//     Term 99 (AT2000-0250)/CC Inputs/Current actual value Ch.3 <-> Data Pointer/CurrentActualValues[2]
//     Term 99 (AT2000-0250)/CC Inputs/Current actual value Ch.4 <-> Data Pointer/CurrentActualValues[3]
//     Term 99 (AT2000-0250)/CC Inputs/Current actual value Ch.5 <-> Data Pointer/CurrentActualValues[4]
//     Term 99 (AT2000-0250)/CC Inputs/Current actual value Ch.6 <-> Data Pointer/CurrentActualValues[5]
//     Term 99 (AT2000-0250)/CC Inputs/Current actual value Ch.7 <-> Data Pointer/CurrentActualValues[6]
//     Term 99 (AT2000-0250)/CC Inputs/Current actual value Ch.8 <-> Data Pointer/CurrentActualValues[7]
//     Term 99 (AT2000-0250)/CC Inputs/Current actual value Ch.9 <-> Data Pointer/CurrentActualValues[8]
//     Term 99 (AT2000-0250)/CC Inputs/Status <-> Data Pointer/Status
//     Term 99 (AT2000-0250)/CC Outputs/Control <-> Data Pointer/Control
//     Term 99 (AT2000-0250)/CC Outputs/Current setpoint value Ch.1 <-> Data Pointer/CurrentSetpointValues[0]
//     Term 99 (AT2000-0250)/CC Outputs/Current setpoint value Ch.10 <-> Data Pointer/CurrentSetpointValues[9]
//     Term 99 (AT2000-0250)/CC Outputs/Current setpoint value Ch.11 <-> Data Pointer/CurrentSetpointValues[10]
//     Term 99 (AT2000-0250)/CC Outputs/Current setpoint value Ch.12 <-> Data Pointer/CurrentSetpointValues[11]
//     Term 99 (AT2000-0250)/CC Outputs/Current setpoint value Ch.13 <-> Data Pointer/CurrentSetpointValues[12]
//     Term 99 (AT2000-0250)/CC Outputs/Current setpoint value Ch.14 <-> Data Pointer/CurrentSetpointValues[13]
//     Term 99 (AT2000-0250)/CC Outputs/Current setpoint value Ch.15 <-> Data Pointer/CurrentSetpointValues[14]
//     Term 99 (AT2000-0250)/CC Outputs/Current setpoint value Ch.2 <-> Data Pointer/CurrentSetpointValues[1]
//     Term 99 (AT2000-0250)/CC Outputs/Current setpoint value Ch.3 <-> Data Pointer/CurrentSetpointValues[2]
//     Term 99 (AT2000-0250)/CC Outputs/Current setpoint value Ch.4 <-> Data Pointer/CurrentSetpointValues[3]
//     Term 99 (AT2000-0250)/CC Outputs/Current setpoint value Ch.5 <-> Data Pointer/CurrentSetpointValues[4]
//     Term 99 (AT2000-0250)/CC Outputs/Current setpoint value Ch.6 <-> Data Pointer/CurrentSetpointValues[5]
//     Term 99 (AT2000-0250)/CC Outputs/Current setpoint value Ch.7 <-> Data Pointer/CurrentSetpointValues[6]
//     Term 99 (AT2000-0250)/CC Outputs/Current setpoint value Ch.8 <-> Data Pointer/CurrentSetpointValues[7]
//     Term 99 (AT2000-0250)/CC Outputs/Current setpoint value Ch.9 <-> Data Pointer/CurrentSetpointValues[8]
//     Term 99 (AT2000-0250)/Term 100 (AT2000-5250)/FB Inputs/Value Channel 01 <-> Data Pointer/RawPositionValues[0]
//     Term 99 (AT2000-0250)/Term 100 (AT2000-5250)/FB Inputs/Value Channel 02 <-> Data Pointer/RawPositionValues[1]
//     Term 99 (AT2000-0250)/Term 100 (AT2000-5250)/FB Inputs/Value Channel 03 <-> Data Pointer/RawPositionValues[2]
//     Term 99 (AT2000-0250)/Term 100 (AT2000-5250)/FB Inputs/Value Channel 04 <-> Data Pointer/RawPositionValues[3]
//     Term 99 (AT2000-0250)/Term 100 (AT2000-5250)/FB Inputs/Value Channel 05 <-> Data Pointer/RawPositionValues[4]
//     Term 99 (AT2000-0250)/Term 100 (AT2000-5250)/FB Inputs/Value Channel 06 <-> Data Pointer/RawPositionValues[5]
//     Term 99 (AT2000-0250)/Term 100 (AT2000-5250)/FB Inputs/Value Channel 07 <-> Data Pointer/RawPositionValues[6]
//     Term 99 (AT2000-0250)/Term 100 (AT2000-5250)/FB Inputs/Value Channel 08 <-> Data Pointer/RawPositionValues[7]
//     Term 99 (AT2000-0250)/Term 100 (AT2000-5250)/FB Inputs/Value Channel 09 <-> Data Pointer/RawPositionValues[8]
//     Term 99 (AT2000-0250)/Term 100 (AT2000-5250)/FB Inputs/Value Channel 10 <-> Data Pointer/RawPositionValues[9]
//     Term 99 (AT2000-0250)/Term 100 (AT2000-5250)/FB Inputs/Value Channel 11 <-> Data Pointer/RawPositionValues[10]
//     Term 99 (AT2000-0250)/Term 100 (AT2000-5250)/FB Inputs/Value Channel 12 <-> Data Pointer/RawPositionValues[11]
//     Term 99 (AT2000-0250)/Term 100 (AT2000-5250)/FB Inputs/Value Channel 13 <-> Data Pointer/RawPositionValues[12]
//     Term 99 (AT2000-0250)/Term 100 (AT2000-5250)/FB Inputs/Value Channel 14 <-> Data Pointer/RawPositionValues[13]
//     Term 99 (AT2000-0250)/Term 100 (AT2000-5250)/FB Inputs/Value Channel 15 <-> Data Pointer/RawPositionValues[14]
//     Term 99 (AT2000-0250)/Term 100 (AT2000-5250)/FB Inputs/Value Channel 16 <-> Data Pointer/RawPositionValues[15]
//     Term 99 (AT2000-0250)/Term 100 (AT2000-5250)/FB Inputs/Value Channel 17 <-> Data Pointer/RawPositionValues[16]
//     Term 99 (AT2000-0250)/Term 100 (AT2000-5250)/FB Inputs/Value Channel 18 <-> Data Pointer/RawPositionValues[17]
//     Term 99 (AT2000-0250)/Term 100 (AT2000-5250)/FB Inputs/Value Channel 19 <-> Data Pointer/RawPositionValues[18]
//     Term 99 (AT2000-0250)/Term 100 (AT2000-5250)/FB Inputs/Value Channel 20 <-> Data Pointer/RawPositionValues[19]
//     Term 99 (AT2000-0250)/Term 100 (AT2000-5250)/FB Inputs/Value Channel 21 <-> Data Pointer/RawPositionValues[20]
//     Term 99 (AT2000-0250)/Term 100 (AT2000-5250)/FB Inputs/Value Channel 22 <-> Data Pointer/RawPositionValues[21]
//     Term 99 (AT2000-0250)/Term 100 (AT2000-5250)/FB Inputs/Value Channel 23 <-> Data Pointer/RawPositionValues[22]
//     Term 99 (AT2000-0250)/Term 100 (AT2000-5250)/FB Inputs/Value Channel 24 <-> Data Pointer/RawPositionValues[23]
//     Term 99 (AT2000-0250)/Term 100 (AT2000-5250)/FB Inputs/Value Channel 25 <-> Data Pointer/RawPositionValues[24]
//     Term 99 (AT2000-0250)/Term 100 (AT2000-5250)/FB Inputs/Value Channel 26 <-> Data Pointer/RawPositionValues[25]
//     Term 99 (AT2000-0250)/Term 100 (AT2000-5250)/FB Inputs/Value Channel 27 <-> Data Pointer/RawPositionValues[26]
//     Term 99 (AT2000-0250)/Term 100 (AT2000-5250)/FB Inputs/Value Channel 28 <-> Data Pointer/RawPositionValues[27]
//     Term 99 (AT2000-0250)/Term 100 (AT2000-5250)/FB Inputs/Value Channel 29 <-> Data Pointer/RawPositionValues[28]
//     Term 99 (AT2000-0250)/Term 100 (AT2000-5250)/FB Inputs/Value Channel 30 <-> Data Pointer/RawPositionValues[29]
//     Term 99 (AT2000-0250)/Term 100 (AT2000-5250)/FB Inputs/Value Channel 31 <-> Data Pointer/RawPositionValues[30]
//     Term 99 (AT2000-0250)/Term 100 (AT2000-5250)/FB Inputs/Value Channel 32 <-> Data Pointer/RawPositionValues[31]
//   Device 23 <-> TcCOM Objects/XTS ProcessingUnit 1/Part 1/Module 51
//     Term 101 (AT2000-0250)/CC Inputs/Current actual value Ch.1 <-> Data Pointer/CurrentActualValues[0]
//     Term 101 (AT2000-0250)/CC Inputs/Current actual value Ch.10 <-> Data Pointer/CurrentActualValues[9]
//     Term 101 (AT2000-0250)/CC Inputs/Current actual value Ch.11 <-> Data Pointer/CurrentActualValues[10]
//     Term 101 (AT2000-0250)/CC Inputs/Current actual value Ch.12 <-> Data Pointer/CurrentActualValues[11]
//     Term 101 (AT2000-0250)/CC Inputs/Current actual value Ch.13 <-> Data Pointer/CurrentActualValues[12]
//     Term 101 (AT2000-0250)/CC Inputs/Current actual value Ch.14 <-> Data Pointer/CurrentActualValues[13]
//     Term 101 (AT2000-0250)/CC Inputs/Current actual value Ch.15 <-> Data Pointer/CurrentActualValues[14]
//     Term 101 (AT2000-0250)/CC Inputs/Current actual value Ch.2 <-> Data Pointer/CurrentActualValues[1]
//     Term 101 (AT2000-0250)/CC Inputs/Current actual value Ch.3 <-> Data Pointer/CurrentActualValues[2]
//     Term 101 (AT2000-0250)/CC Inputs/Current actual value Ch.4 <-> Data Pointer/CurrentActualValues[3]
//     Term 101 (AT2000-0250)/CC Inputs/Current actual value Ch.5 <-> Data Pointer/CurrentActualValues[4]
//     Term 101 (AT2000-0250)/CC Inputs/Current actual value Ch.6 <-> Data Pointer/CurrentActualValues[5]
//     Term 101 (AT2000-0250)/CC Inputs/Current actual value Ch.7 <-> Data Pointer/CurrentActualValues[6]
//     Term 101 (AT2000-0250)/CC Inputs/Current actual value Ch.8 <-> Data Pointer/CurrentActualValues[7]
//     Term 101 (AT2000-0250)/CC Inputs/Current actual value Ch.9 <-> Data Pointer/CurrentActualValues[8]
//     Term 101 (AT2000-0250)/CC Inputs/Status <-> Data Pointer/Status
//     Term 101 (AT2000-0250)/CC Outputs/Control <-> Data Pointer/Control
//     Term 101 (AT2000-0250)/CC Outputs/Current setpoint value Ch.1 <-> Data Pointer/CurrentSetpointValues[0]
//     Term 101 (AT2000-0250)/CC Outputs/Current setpoint value Ch.10 <-> Data Pointer/CurrentSetpointValues[9]
//     Term 101 (AT2000-0250)/CC Outputs/Current setpoint value Ch.11 <-> Data Pointer/CurrentSetpointValues[10]
//     Term 101 (AT2000-0250)/CC Outputs/Current setpoint value Ch.12 <-> Data Pointer/CurrentSetpointValues[11]
//     Term 101 (AT2000-0250)/CC Outputs/Current setpoint value Ch.13 <-> Data Pointer/CurrentSetpointValues[12]
//     Term 101 (AT2000-0250)/CC Outputs/Current setpoint value Ch.14 <-> Data Pointer/CurrentSetpointValues[13]
//     Term 101 (AT2000-0250)/CC Outputs/Current setpoint value Ch.15 <-> Data Pointer/CurrentSetpointValues[14]
//     Term 101 (AT2000-0250)/CC Outputs/Current setpoint value Ch.2 <-> Data Pointer/CurrentSetpointValues[1]
//     Term 101 (AT2000-0250)/CC Outputs/Current setpoint value Ch.3 <-> Data Pointer/CurrentSetpointValues[2]
//     Term 101 (AT2000-0250)/CC Outputs/Current setpoint value Ch.4 <-> Data Pointer/CurrentSetpointValues[3]
//     Term 101 (AT2000-0250)/CC Outputs/Current setpoint value Ch.5 <-> Data Pointer/CurrentSetpointValues[4]
//     Term 101 (AT2000-0250)/CC Outputs/Current setpoint value Ch.6 <-> Data Pointer/CurrentSetpointValues[5]
//     Term 101 (AT2000-0250)/CC Outputs/Current setpoint value Ch.7 <-> Data Pointer/CurrentSetpointValues[6]
//     Term 101 (AT2000-0250)/CC Outputs/Current setpoint value Ch.8 <-> Data Pointer/CurrentSetpointValues[7]
//     Term 101 (AT2000-0250)/CC Outputs/Current setpoint value Ch.9 <-> Data Pointer/CurrentSetpointValues[8]
//     Term 101 (AT2000-0250)/Term 102 (AT2000-5250)/FB Inputs/Value Channel 01 <-> Data Pointer/RawPositionValues[0]
//     Term 101 (AT2000-0250)/Term 102 (AT2000-5250)/FB Inputs/Value Channel 02 <-> Data Pointer/RawPositionValues[1]
//     Term 101 (AT2000-0250)/Term 102 (AT2000-5250)/FB Inputs/Value Channel 03 <-> Data Pointer/RawPositionValues[2]
//     Term 101 (AT2000-0250)/Term 102 (AT2000-5250)/FB Inputs/Value Channel 04 <-> Data Pointer/RawPositionValues[3]
//     Term 101 (AT2000-0250)/Term 102 (AT2000-5250)/FB Inputs/Value Channel 05 <-> Data Pointer/RawPositionValues[4]
//     Term 101 (AT2000-0250)/Term 102 (AT2000-5250)/FB Inputs/Value Channel 06 <-> Data Pointer/RawPositionValues[5]
//     Term 101 (AT2000-0250)/Term 102 (AT2000-5250)/FB Inputs/Value Channel 07 <-> Data Pointer/RawPositionValues[6]
//     Term 101 (AT2000-0250)/Term 102 (AT2000-5250)/FB Inputs/Value Channel 08 <-> Data Pointer/RawPositionValues[7]
//     Term 101 (AT2000-0250)/Term 102 (AT2000-5250)/FB Inputs/Value Channel 09 <-> Data Pointer/RawPositionValues[8]
//     Term 101 (AT2000-0250)/Term 102 (AT2000-5250)/FB Inputs/Value Channel 10 <-> Data Pointer/RawPositionValues[9]
//     Term 101 (AT2000-0250)/Term 102 (AT2000-5250)/FB Inputs/Value Channel 11 <-> Data Pointer/RawPositionValues[10]
//     Term 101 (AT2000-0250)/Term 102 (AT2000-5250)/FB Inputs/Value Channel 12 <-> Data Pointer/RawPositionValues[11]
//     Term 101 (AT2000-0250)/Term 102 (AT2000-5250)/FB Inputs/Value Channel 13 <-> Data Pointer/RawPositionValues[12]
//     Term 101 (AT2000-0250)/Term 102 (AT2000-5250)/FB Inputs/Value Channel 14 <-> Data Pointer/RawPositionValues[13]
//     Term 101 (AT2000-0250)/Term 102 (AT2000-5250)/FB Inputs/Value Channel 15 <-> Data Pointer/RawPositionValues[14]
//     Term 101 (AT2000-0250)/Term 102 (AT2000-5250)/FB Inputs/Value Channel 16 <-> Data Pointer/RawPositionValues[15]
//     Term 101 (AT2000-0250)/Term 102 (AT2000-5250)/FB Inputs/Value Channel 17 <-> Data Pointer/RawPositionValues[16]
//     Term 101 (AT2000-0250)/Term 102 (AT2000-5250)/FB Inputs/Value Channel 18 <-> Data Pointer/RawPositionValues[17]
//     Term 101 (AT2000-0250)/Term 102 (AT2000-5250)/FB Inputs/Value Channel 19 <-> Data Pointer/RawPositionValues[18]
//     Term 101 (AT2000-0250)/Term 102 (AT2000-5250)/FB Inputs/Value Channel 20 <-> Data Pointer/RawPositionValues[19]
//     Term 101 (AT2000-0250)/Term 102 (AT2000-5250)/FB Inputs/Value Channel 21 <-> Data Pointer/RawPositionValues[20]
//     Term 101 (AT2000-0250)/Term 102 (AT2000-5250)/FB Inputs/Value Channel 22 <-> Data Pointer/RawPositionValues[21]
//     Term 101 (AT2000-0250)/Term 102 (AT2000-5250)/FB Inputs/Value Channel 23 <-> Data Pointer/RawPositionValues[22]
//     Term 101 (AT2000-0250)/Term 102 (AT2000-5250)/FB Inputs/Value Channel 24 <-> Data Pointer/RawPositionValues[23]
//     Term 101 (AT2000-0250)/Term 102 (AT2000-5250)/FB Inputs/Value Channel 25 <-> Data Pointer/RawPositionValues[24]
//     Term 101 (AT2000-0250)/Term 102 (AT2000-5250)/FB Inputs/Value Channel 26 <-> Data Pointer/RawPositionValues[25]
//     Term 101 (AT2000-0250)/Term 102 (AT2000-5250)/FB Inputs/Value Channel 27 <-> Data Pointer/RawPositionValues[26]
//     Term 101 (AT2000-0250)/Term 102 (AT2000-5250)/FB Inputs/Value Channel 28 <-> Data Pointer/RawPositionValues[27]
//     Term 101 (AT2000-0250)/Term 102 (AT2000-5250)/FB Inputs/Value Channel 29 <-> Data Pointer/RawPositionValues[28]
//     Term 101 (AT2000-0250)/Term 102 (AT2000-5250)/FB Inputs/Value Channel 30 <-> Data Pointer/RawPositionValues[29]
//     Term 101 (AT2000-0250)/Term 102 (AT2000-5250)/FB Inputs/Value Channel 31 <-> Data Pointer/RawPositionValues[30]
//     Term 101 (AT2000-0250)/Term 102 (AT2000-5250)/FB Inputs/Value Channel 32 <-> Data Pointer/RawPositionValues[31]
//   Device 23 <-> TcCOM Objects/XTS ProcessingUnit 1/Part 1/Module 52
//     Term 103 (AT2000-0250)/CC Inputs/Current actual value Ch.1 <-> Data Pointer/CurrentActualValues[0]
//     Term 103 (AT2000-0250)/CC Inputs/Current actual value Ch.10 <-> Data Pointer/CurrentActualValues[9]
//     Term 103 (AT2000-0250)/CC Inputs/Current actual value Ch.11 <-> Data Pointer/CurrentActualValues[10]
//     Term 103 (AT2000-0250)/CC Inputs/Current actual value Ch.12 <-> Data Pointer/CurrentActualValues[11]
//     Term 103 (AT2000-0250)/CC Inputs/Current actual value Ch.13 <-> Data Pointer/CurrentActualValues[12]
//     Term 103 (AT2000-0250)/CC Inputs/Current actual value Ch.14 <-> Data Pointer/CurrentActualValues[13]
//     Term 103 (AT2000-0250)/CC Inputs/Current actual value Ch.15 <-> Data Pointer/CurrentActualValues[14]
//     Term 103 (AT2000-0250)/CC Inputs/Current actual value Ch.2 <-> Data Pointer/CurrentActualValues[1]
//     Term 103 (AT2000-0250)/CC Inputs/Current actual value Ch.3 <-> Data Pointer/CurrentActualValues[2]
//     Term 103 (AT2000-0250)/CC Inputs/Current actual value Ch.4 <-> Data Pointer/CurrentActualValues[3]
//     Term 103 (AT2000-0250)/CC Inputs/Current actual value Ch.5 <-> Data Pointer/CurrentActualValues[4]
//     Term 103 (AT2000-0250)/CC Inputs/Current actual value Ch.6 <-> Data Pointer/CurrentActualValues[5]
//     Term 103 (AT2000-0250)/CC Inputs/Current actual value Ch.7 <-> Data Pointer/CurrentActualValues[6]
//     Term 103 (AT2000-0250)/CC Inputs/Current actual value Ch.8 <-> Data Pointer/CurrentActualValues[7]
//     Term 103 (AT2000-0250)/CC Inputs/Current actual value Ch.9 <-> Data Pointer/CurrentActualValues[8]
//     Term 103 (AT2000-0250)/CC Inputs/Status <-> Data Pointer/Status
//     Term 103 (AT2000-0250)/CC Outputs/Control <-> Data Pointer/Control
//     Term 103 (AT2000-0250)/CC Outputs/Current setpoint value Ch.1 <-> Data Pointer/CurrentSetpointValues[0]
//     Term 103 (AT2000-0250)/CC Outputs/Current setpoint value Ch.10 <-> Data Pointer/CurrentSetpointValues[9]
//     Term 103 (AT2000-0250)/CC Outputs/Current setpoint value Ch.11 <-> Data Pointer/CurrentSetpointValues[10]
//     Term 103 (AT2000-0250)/CC Outputs/Current setpoint value Ch.12 <-> Data Pointer/CurrentSetpointValues[11]
//     Term 103 (AT2000-0250)/CC Outputs/Current setpoint value Ch.13 <-> Data Pointer/CurrentSetpointValues[12]
//     Term 103 (AT2000-0250)/CC Outputs/Current setpoint value Ch.14 <-> Data Pointer/CurrentSetpointValues[13]
//     Term 103 (AT2000-0250)/CC Outputs/Current setpoint value Ch.15 <-> Data Pointer/CurrentSetpointValues[14]
//     Term 103 (AT2000-0250)/CC Outputs/Current setpoint value Ch.2 <-> Data Pointer/CurrentSetpointValues[1]
//     Term 103 (AT2000-0250)/CC Outputs/Current setpoint value Ch.3 <-> Data Pointer/CurrentSetpointValues[2]
//     Term 103 (AT2000-0250)/CC Outputs/Current setpoint value Ch.4 <-> Data Pointer/CurrentSetpointValues[3]
//     Term 103 (AT2000-0250)/CC Outputs/Current setpoint value Ch.5 <-> Data Pointer/CurrentSetpointValues[4]
//     Term 103 (AT2000-0250)/CC Outputs/Current setpoint value Ch.6 <-> Data Pointer/CurrentSetpointValues[5]
//     Term 103 (AT2000-0250)/CC Outputs/Current setpoint value Ch.7 <-> Data Pointer/CurrentSetpointValues[6]
//     Term 103 (AT2000-0250)/CC Outputs/Current setpoint value Ch.8 <-> Data Pointer/CurrentSetpointValues[7]
//     Term 103 (AT2000-0250)/CC Outputs/Current setpoint value Ch.9 <-> Data Pointer/CurrentSetpointValues[8]
//     Term 103 (AT2000-0250)/Term 104 (AT2000-5250)/FB Inputs/Value Channel 01 <-> Data Pointer/RawPositionValues[0]
//     Term 103 (AT2000-0250)/Term 104 (AT2000-5250)/FB Inputs/Value Channel 02 <-> Data Pointer/RawPositionValues[1]
//     Term 103 (AT2000-0250)/Term 104 (AT2000-5250)/FB Inputs/Value Channel 03 <-> Data Pointer/RawPositionValues[2]
//     Term 103 (AT2000-0250)/Term 104 (AT2000-5250)/FB Inputs/Value Channel 04 <-> Data Pointer/RawPositionValues[3]
//     Term 103 (AT2000-0250)/Term 104 (AT2000-5250)/FB Inputs/Value Channel 05 <-> Data Pointer/RawPositionValues[4]
//     Term 103 (AT2000-0250)/Term 104 (AT2000-5250)/FB Inputs/Value Channel 06 <-> Data Pointer/RawPositionValues[5]
//     Term 103 (AT2000-0250)/Term 104 (AT2000-5250)/FB Inputs/Value Channel 07 <-> Data Pointer/RawPositionValues[6]
//     Term 103 (AT2000-0250)/Term 104 (AT2000-5250)/FB Inputs/Value Channel 08 <-> Data Pointer/RawPositionValues[7]
//     Term 103 (AT2000-0250)/Term 104 (AT2000-5250)/FB Inputs/Value Channel 09 <-> Data Pointer/RawPositionValues[8]
//     Term 103 (AT2000-0250)/Term 104 (AT2000-5250)/FB Inputs/Value Channel 10 <-> Data Pointer/RawPositionValues[9]
//     Term 103 (AT2000-0250)/Term 104 (AT2000-5250)/FB Inputs/Value Channel 11 <-> Data Pointer/RawPositionValues[10]
//     Term 103 (AT2000-0250)/Term 104 (AT2000-5250)/FB Inputs/Value Channel 12 <-> Data Pointer/RawPositionValues[11]
//     Term 103 (AT2000-0250)/Term 104 (AT2000-5250)/FB Inputs/Value Channel 13 <-> Data Pointer/RawPositionValues[12]
//     Term 103 (AT2000-0250)/Term 104 (AT2000-5250)/FB Inputs/Value Channel 14 <-> Data Pointer/RawPositionValues[13]
//     Term 103 (AT2000-0250)/Term 104 (AT2000-5250)/FB Inputs/Value Channel 15 <-> Data Pointer/RawPositionValues[14]
//     Term 103 (AT2000-0250)/Term 104 (AT2000-5250)/FB Inputs/Value Channel 16 <-> Data Pointer/RawPositionValues[15]
//     Term 103 (AT2000-0250)/Term 104 (AT2000-5250)/FB Inputs/Value Channel 17 <-> Data Pointer/RawPositionValues[16]
//     Term 103 (AT2000-0250)/Term 104 (AT2000-5250)/FB Inputs/Value Channel 18 <-> Data Pointer/RawPositionValues[17]
//     Term 103 (AT2000-0250)/Term 104 (AT2000-5250)/FB Inputs/Value Channel 19 <-> Data Pointer/RawPositionValues[18]
//     Term 103 (AT2000-0250)/Term 104 (AT2000-5250)/FB Inputs/Value Channel 20 <-> Data Pointer/RawPositionValues[19]
//     Term 103 (AT2000-0250)/Term 104 (AT2000-5250)/FB Inputs/Value Channel 21 <-> Data Pointer/RawPositionValues[20]
//     Term 103 (AT2000-0250)/Term 104 (AT2000-5250)/FB Inputs/Value Channel 22 <-> Data Pointer/RawPositionValues[21]
//     Term 103 (AT2000-0250)/Term 104 (AT2000-5250)/FB Inputs/Value Channel 23 <-> Data Pointer/RawPositionValues[22]
//     Term 103 (AT2000-0250)/Term 104 (AT2000-5250)/FB Inputs/Value Channel 24 <-> Data Pointer/RawPositionValues[23]
//     Term 103 (AT2000-0250)/Term 104 (AT2000-5250)/FB Inputs/Value Channel 25 <-> Data Pointer/RawPositionValues[24]
//     Term 103 (AT2000-0250)/Term 104 (AT2000-5250)/FB Inputs/Value Channel 26 <-> Data Pointer/RawPositionValues[25]
//     Term 103 (AT2000-0250)/Term 104 (AT2000-5250)/FB Inputs/Value Channel 27 <-> Data Pointer/RawPositionValues[26]
//     Term 103 (AT2000-0250)/Term 104 (AT2000-5250)/FB Inputs/Value Channel 28 <-> Data Pointer/RawPositionValues[27]
//     Term 103 (AT2000-0250)/Term 104 (AT2000-5250)/FB Inputs/Value Channel 29 <-> Data Pointer/RawPositionValues[28]
//     Term 103 (AT2000-0250)/Term 104 (AT2000-5250)/FB Inputs/Value Channel 30 <-> Data Pointer/RawPositionValues[29]
//     Term 103 (AT2000-0250)/Term 104 (AT2000-5250)/FB Inputs/Value Channel 31 <-> Data Pointer/RawPositionValues[30]
//     Term 103 (AT2000-0250)/Term 104 (AT2000-5250)/FB Inputs/Value Channel 32 <-> Data Pointer/RawPositionValues[31]
//   Device 23 <-> TcCOM Objects/XTS ProcessingUnit 1/Part 1/Module 53
//     Term 105 (AT2000-0250)/CC Inputs/Current actual value Ch.1 <-> Data Pointer/CurrentActualValues[0]
//     Term 105 (AT2000-0250)/CC Inputs/Current actual value Ch.10 <-> Data Pointer/CurrentActualValues[9]
//     Term 105 (AT2000-0250)/CC Inputs/Current actual value Ch.11 <-> Data Pointer/CurrentActualValues[10]
//     Term 105 (AT2000-0250)/CC Inputs/Current actual value Ch.12 <-> Data Pointer/CurrentActualValues[11]
//     Term 105 (AT2000-0250)/CC Inputs/Current actual value Ch.13 <-> Data Pointer/CurrentActualValues[12]
//     Term 105 (AT2000-0250)/CC Inputs/Current actual value Ch.14 <-> Data Pointer/CurrentActualValues[13]
//     Term 105 (AT2000-0250)/CC Inputs/Current actual value Ch.15 <-> Data Pointer/CurrentActualValues[14]
//     Term 105 (AT2000-0250)/CC Inputs/Current actual value Ch.2 <-> Data Pointer/CurrentActualValues[1]
//     Term 105 (AT2000-0250)/CC Inputs/Current actual value Ch.3 <-> Data Pointer/CurrentActualValues[2]
//     Term 105 (AT2000-0250)/CC Inputs/Current actual value Ch.4 <-> Data Pointer/CurrentActualValues[3]
//     Term 105 (AT2000-0250)/CC Inputs/Current actual value Ch.5 <-> Data Pointer/CurrentActualValues[4]
//     Term 105 (AT2000-0250)/CC Inputs/Current actual value Ch.6 <-> Data Pointer/CurrentActualValues[5]
//     Term 105 (AT2000-0250)/CC Inputs/Current actual value Ch.7 <-> Data Pointer/CurrentActualValues[6]
//     Term 105 (AT2000-0250)/CC Inputs/Current actual value Ch.8 <-> Data Pointer/CurrentActualValues[7]
//     Term 105 (AT2000-0250)/CC Inputs/Current actual value Ch.9 <-> Data Pointer/CurrentActualValues[8]
//     Term 105 (AT2000-0250)/CC Inputs/Status <-> Data Pointer/Status
//     Term 105 (AT2000-0250)/CC Outputs/Control <-> Data Pointer/Control
//     Term 105 (AT2000-0250)/CC Outputs/Current setpoint value Ch.1 <-> Data Pointer/CurrentSetpointValues[0]
//     Term 105 (AT2000-0250)/CC Outputs/Current setpoint value Ch.10 <-> Data Pointer/CurrentSetpointValues[9]
//     Term 105 (AT2000-0250)/CC Outputs/Current setpoint value Ch.11 <-> Data Pointer/CurrentSetpointValues[10]
//     Term 105 (AT2000-0250)/CC Outputs/Current setpoint value Ch.12 <-> Data Pointer/CurrentSetpointValues[11]
//     Term 105 (AT2000-0250)/CC Outputs/Current setpoint value Ch.13 <-> Data Pointer/CurrentSetpointValues[12]
//     Term 105 (AT2000-0250)/CC Outputs/Current setpoint value Ch.14 <-> Data Pointer/CurrentSetpointValues[13]
//     Term 105 (AT2000-0250)/CC Outputs/Current setpoint value Ch.15 <-> Data Pointer/CurrentSetpointValues[14]
//     Term 105 (AT2000-0250)/CC Outputs/Current setpoint value Ch.2 <-> Data Pointer/CurrentSetpointValues[1]
//     Term 105 (AT2000-0250)/CC Outputs/Current setpoint value Ch.3 <-> Data Pointer/CurrentSetpointValues[2]
//     Term 105 (AT2000-0250)/CC Outputs/Current setpoint value Ch.4 <-> Data Pointer/CurrentSetpointValues[3]
//     Term 105 (AT2000-0250)/CC Outputs/Current setpoint value Ch.5 <-> Data Pointer/CurrentSetpointValues[4]
//     Term 105 (AT2000-0250)/CC Outputs/Current setpoint value Ch.6 <-> Data Pointer/CurrentSetpointValues[5]
//     Term 105 (AT2000-0250)/CC Outputs/Current setpoint value Ch.7 <-> Data Pointer/CurrentSetpointValues[6]
//     Term 105 (AT2000-0250)/CC Outputs/Current setpoint value Ch.8 <-> Data Pointer/CurrentSetpointValues[7]
//     Term 105 (AT2000-0250)/CC Outputs/Current setpoint value Ch.9 <-> Data Pointer/CurrentSetpointValues[8]
//     Term 105 (AT2000-0250)/Term 106 (AT2000-5250)/FB Inputs/Value Channel 01 <-> Data Pointer/RawPositionValues[0]
//     Term 105 (AT2000-0250)/Term 106 (AT2000-5250)/FB Inputs/Value Channel 02 <-> Data Pointer/RawPositionValues[1]
//     Term 105 (AT2000-0250)/Term 106 (AT2000-5250)/FB Inputs/Value Channel 03 <-> Data Pointer/RawPositionValues[2]
//     Term 105 (AT2000-0250)/Term 106 (AT2000-5250)/FB Inputs/Value Channel 04 <-> Data Pointer/RawPositionValues[3]
//     Term 105 (AT2000-0250)/Term 106 (AT2000-5250)/FB Inputs/Value Channel 05 <-> Data Pointer/RawPositionValues[4]
//     Term 105 (AT2000-0250)/Term 106 (AT2000-5250)/FB Inputs/Value Channel 06 <-> Data Pointer/RawPositionValues[5]
//     Term 105 (AT2000-0250)/Term 106 (AT2000-5250)/FB Inputs/Value Channel 07 <-> Data Pointer/RawPositionValues[6]
//     Term 105 (AT2000-0250)/Term 106 (AT2000-5250)/FB Inputs/Value Channel 08 <-> Data Pointer/RawPositionValues[7]
//     Term 105 (AT2000-0250)/Term 106 (AT2000-5250)/FB Inputs/Value Channel 09 <-> Data Pointer/RawPositionValues[8]
//     Term 105 (AT2000-0250)/Term 106 (AT2000-5250)/FB Inputs/Value Channel 10 <-> Data Pointer/RawPositionValues[9]
//     Term 105 (AT2000-0250)/Term 106 (AT2000-5250)/FB Inputs/Value Channel 11 <-> Data Pointer/RawPositionValues[10]
//     Term 105 (AT2000-0250)/Term 106 (AT2000-5250)/FB Inputs/Value Channel 12 <-> Data Pointer/RawPositionValues[11]
//     Term 105 (AT2000-0250)/Term 106 (AT2000-5250)/FB Inputs/Value Channel 13 <-> Data Pointer/RawPositionValues[12]
//     Term 105 (AT2000-0250)/Term 106 (AT2000-5250)/FB Inputs/Value Channel 14 <-> Data Pointer/RawPositionValues[13]
//     Term 105 (AT2000-0250)/Term 106 (AT2000-5250)/FB Inputs/Value Channel 15 <-> Data Pointer/RawPositionValues[14]
//     Term 105 (AT2000-0250)/Term 106 (AT2000-5250)/FB Inputs/Value Channel 16 <-> Data Pointer/RawPositionValues[15]
//     Term 105 (AT2000-0250)/Term 106 (AT2000-5250)/FB Inputs/Value Channel 17 <-> Data Pointer/RawPositionValues[16]
//     Term 105 (AT2000-0250)/Term 106 (AT2000-5250)/FB Inputs/Value Channel 18 <-> Data Pointer/RawPositionValues[17]
//     Term 105 (AT2000-0250)/Term 106 (AT2000-5250)/FB Inputs/Value Channel 19 <-> Data Pointer/RawPositionValues[18]
//     Term 105 (AT2000-0250)/Term 106 (AT2000-5250)/FB Inputs/Value Channel 20 <-> Data Pointer/RawPositionValues[19]
//     Term 105 (AT2000-0250)/Term 106 (AT2000-5250)/FB Inputs/Value Channel 21 <-> Data Pointer/RawPositionValues[20]
//     Term 105 (AT2000-0250)/Term 106 (AT2000-5250)/FB Inputs/Value Channel 22 <-> Data Pointer/RawPositionValues[21]
//     Term 105 (AT2000-0250)/Term 106 (AT2000-5250)/FB Inputs/Value Channel 23 <-> Data Pointer/RawPositionValues[22]
//     Term 105 (AT2000-0250)/Term 106 (AT2000-5250)/FB Inputs/Value Channel 24 <-> Data Pointer/RawPositionValues[23]
//     Term 105 (AT2000-0250)/Term 106 (AT2000-5250)/FB Inputs/Value Channel 25 <-> Data Pointer/RawPositionValues[24]
//     Term 105 (AT2000-0250)/Term 106 (AT2000-5250)/FB Inputs/Value Channel 26 <-> Data Pointer/RawPositionValues[25]
//     Term 105 (AT2000-0250)/Term 106 (AT2000-5250)/FB Inputs/Value Channel 27 <-> Data Pointer/RawPositionValues[26]
//     Term 105 (AT2000-0250)/Term 106 (AT2000-5250)/FB Inputs/Value Channel 28 <-> Data Pointer/RawPositionValues[27]
//     Term 105 (AT2000-0250)/Term 106 (AT2000-5250)/FB Inputs/Value Channel 29 <-> Data Pointer/RawPositionValues[28]
//     Term 105 (AT2000-0250)/Term 106 (AT2000-5250)/FB Inputs/Value Channel 30 <-> Data Pointer/RawPositionValues[29]
//     Term 105 (AT2000-0250)/Term 106 (AT2000-5250)/FB Inputs/Value Channel 31 <-> Data Pointer/RawPositionValues[30]
//     Term 105 (AT2000-0250)/Term 106 (AT2000-5250)/FB Inputs/Value Channel 32 <-> Data Pointer/RawPositionValues[31]
//   Device 23 <-> TcCOM Objects/XTS ProcessingUnit 1/Part 1/Module 54
//     Term 107 (AT2000-0250)/CC Inputs/Current actual value Ch.1 <-> Data Pointer/CurrentActualValues[0]
//     Term 107 (AT2000-0250)/CC Inputs/Current actual value Ch.10 <-> Data Pointer/CurrentActualValues[9]
//     Term 107 (AT2000-0250)/CC Inputs/Current actual value Ch.11 <-> Data Pointer/CurrentActualValues[10]
//     Term 107 (AT2000-0250)/CC Inputs/Current actual value Ch.12 <-> Data Pointer/CurrentActualValues[11]
//     Term 107 (AT2000-0250)/CC Inputs/Current actual value Ch.13 <-> Data Pointer/CurrentActualValues[12]
//     Term 107 (AT2000-0250)/CC Inputs/Current actual value Ch.14 <-> Data Pointer/CurrentActualValues[13]
//     Term 107 (AT2000-0250)/CC Inputs/Current actual value Ch.15 <-> Data Pointer/CurrentActualValues[14]
//     Term 107 (AT2000-0250)/CC Inputs/Current actual value Ch.2 <-> Data Pointer/CurrentActualValues[1]
//     Term 107 (AT2000-0250)/CC Inputs/Current actual value Ch.3 <-> Data Pointer/CurrentActualValues[2]
//     Term 107 (AT2000-0250)/CC Inputs/Current actual value Ch.4 <-> Data Pointer/CurrentActualValues[3]
//     Term 107 (AT2000-0250)/CC Inputs/Current actual value Ch.5 <-> Data Pointer/CurrentActualValues[4]
//     Term 107 (AT2000-0250)/CC Inputs/Current actual value Ch.6 <-> Data Pointer/CurrentActualValues[5]
//     Term 107 (AT2000-0250)/CC Inputs/Current actual value Ch.7 <-> Data Pointer/CurrentActualValues[6]
//     Term 107 (AT2000-0250)/CC Inputs/Current actual value Ch.8 <-> Data Pointer/CurrentActualValues[7]
//     Term 107 (AT2000-0250)/CC Inputs/Current actual value Ch.9 <-> Data Pointer/CurrentActualValues[8]
//     Term 107 (AT2000-0250)/CC Inputs/Status <-> Data Pointer/Status
//     Term 107 (AT2000-0250)/CC Outputs/Control <-> Data Pointer/Control
//     Term 107 (AT2000-0250)/CC Outputs/Current setpoint value Ch.1 <-> Data Pointer/CurrentSetpointValues[0]
//     Term 107 (AT2000-0250)/CC Outputs/Current setpoint value Ch.10 <-> Data Pointer/CurrentSetpointValues[9]
//     Term 107 (AT2000-0250)/CC Outputs/Current setpoint value Ch.11 <-> Data Pointer/CurrentSetpointValues[10]
//     Term 107 (AT2000-0250)/CC Outputs/Current setpoint value Ch.12 <-> Data Pointer/CurrentSetpointValues[11]
//     Term 107 (AT2000-0250)/CC Outputs/Current setpoint value Ch.13 <-> Data Pointer/CurrentSetpointValues[12]
//     Term 107 (AT2000-0250)/CC Outputs/Current setpoint value Ch.14 <-> Data Pointer/CurrentSetpointValues[13]
//     Term 107 (AT2000-0250)/CC Outputs/Current setpoint value Ch.15 <-> Data Pointer/CurrentSetpointValues[14]
//     Term 107 (AT2000-0250)/CC Outputs/Current setpoint value Ch.2 <-> Data Pointer/CurrentSetpointValues[1]
//     Term 107 (AT2000-0250)/CC Outputs/Current setpoint value Ch.3 <-> Data Pointer/CurrentSetpointValues[2]
//     Term 107 (AT2000-0250)/CC Outputs/Current setpoint value Ch.4 <-> Data Pointer/CurrentSetpointValues[3]
//     Term 107 (AT2000-0250)/CC Outputs/Current setpoint value Ch.5 <-> Data Pointer/CurrentSetpointValues[4]
//     Term 107 (AT2000-0250)/CC Outputs/Current setpoint value Ch.6 <-> Data Pointer/CurrentSetpointValues[5]
//     Term 107 (AT2000-0250)/CC Outputs/Current setpoint value Ch.7 <-> Data Pointer/CurrentSetpointValues[6]
//     Term 107 (AT2000-0250)/CC Outputs/Current setpoint value Ch.8 <-> Data Pointer/CurrentSetpointValues[7]
//     Term 107 (AT2000-0250)/CC Outputs/Current setpoint value Ch.9 <-> Data Pointer/CurrentSetpointValues[8]
//     Term 107 (AT2000-0250)/Term 108 (AT2000-5250)/FB Inputs/Value Channel 01 <-> Data Pointer/RawPositionValues[0]
//     Term 107 (AT2000-0250)/Term 108 (AT2000-5250)/FB Inputs/Value Channel 02 <-> Data Pointer/RawPositionValues[1]
//     Term 107 (AT2000-0250)/Term 108 (AT2000-5250)/FB Inputs/Value Channel 03 <-> Data Pointer/RawPositionValues[2]
//     Term 107 (AT2000-0250)/Term 108 (AT2000-5250)/FB Inputs/Value Channel 04 <-> Data Pointer/RawPositionValues[3]
//     Term 107 (AT2000-0250)/Term 108 (AT2000-5250)/FB Inputs/Value Channel 05 <-> Data Pointer/RawPositionValues[4]
//     Term 107 (AT2000-0250)/Term 108 (AT2000-5250)/FB Inputs/Value Channel 06 <-> Data Pointer/RawPositionValues[5]
//     Term 107 (AT2000-0250)/Term 108 (AT2000-5250)/FB Inputs/Value Channel 07 <-> Data Pointer/RawPositionValues[6]
//     Term 107 (AT2000-0250)/Term 108 (AT2000-5250)/FB Inputs/Value Channel 08 <-> Data Pointer/RawPositionValues[7]
//     Term 107 (AT2000-0250)/Term 108 (AT2000-5250)/FB Inputs/Value Channel 09 <-> Data Pointer/RawPositionValues[8]
//     Term 107 (AT2000-0250)/Term 108 (AT2000-5250)/FB Inputs/Value Channel 10 <-> Data Pointer/RawPositionValues[9]
//     Term 107 (AT2000-0250)/Term 108 (AT2000-5250)/FB Inputs/Value Channel 11 <-> Data Pointer/RawPositionValues[10]
//     Term 107 (AT2000-0250)/Term 108 (AT2000-5250)/FB Inputs/Value Channel 12 <-> Data Pointer/RawPositionValues[11]
//     Term 107 (AT2000-0250)/Term 108 (AT2000-5250)/FB Inputs/Value Channel 13 <-> Data Pointer/RawPositionValues[12]
//     Term 107 (AT2000-0250)/Term 108 (AT2000-5250)/FB Inputs/Value Channel 14 <-> Data Pointer/RawPositionValues[13]
//     Term 107 (AT2000-0250)/Term 108 (AT2000-5250)/FB Inputs/Value Channel 15 <-> Data Pointer/RawPositionValues[14]
//     Term 107 (AT2000-0250)/Term 108 (AT2000-5250)/FB Inputs/Value Channel 16 <-> Data Pointer/RawPositionValues[15]
//     Term 107 (AT2000-0250)/Term 108 (AT2000-5250)/FB Inputs/Value Channel 17 <-> Data Pointer/RawPositionValues[16]
//     Term 107 (AT2000-0250)/Term 108 (AT2000-5250)/FB Inputs/Value Channel 18 <-> Data Pointer/RawPositionValues[17]
//     Term 107 (AT2000-0250)/Term 108 (AT2000-5250)/FB Inputs/Value Channel 19 <-> Data Pointer/RawPositionValues[18]
//     Term 107 (AT2000-0250)/Term 108 (AT2000-5250)/FB Inputs/Value Channel 20 <-> Data Pointer/RawPositionValues[19]
//     Term 107 (AT2000-0250)/Term 108 (AT2000-5250)/FB Inputs/Value Channel 21 <-> Data Pointer/RawPositionValues[20]
//     Term 107 (AT2000-0250)/Term 108 (AT2000-5250)/FB Inputs/Value Channel 22 <-> Data Pointer/RawPositionValues[21]
//     Term 107 (AT2000-0250)/Term 108 (AT2000-5250)/FB Inputs/Value Channel 23 <-> Data Pointer/RawPositionValues[22]
//     Term 107 (AT2000-0250)/Term 108 (AT2000-5250)/FB Inputs/Value Channel 24 <-> Data Pointer/RawPositionValues[23]
//     Term 107 (AT2000-0250)/Term 108 (AT2000-5250)/FB Inputs/Value Channel 25 <-> Data Pointer/RawPositionValues[24]
//     Term 107 (AT2000-0250)/Term 108 (AT2000-5250)/FB Inputs/Value Channel 26 <-> Data Pointer/RawPositionValues[25]
//     Term 107 (AT2000-0250)/Term 108 (AT2000-5250)/FB Inputs/Value Channel 27 <-> Data Pointer/RawPositionValues[26]
//     Term 107 (AT2000-0250)/Term 108 (AT2000-5250)/FB Inputs/Value Channel 28 <-> Data Pointer/RawPositionValues[27]
//     Term 107 (AT2000-0250)/Term 108 (AT2000-5250)/FB Inputs/Value Channel 29 <-> Data Pointer/RawPositionValues[28]
//     Term 107 (AT2000-0250)/Term 108 (AT2000-5250)/FB Inputs/Value Channel 30 <-> Data Pointer/RawPositionValues[29]
//     Term 107 (AT2000-0250)/Term 108 (AT2000-5250)/FB Inputs/Value Channel 31 <-> Data Pointer/RawPositionValues[30]
//     Term 107 (AT2000-0250)/Term 108 (AT2000-5250)/FB Inputs/Value Channel 32 <-> Data Pointer/RawPositionValues[31]
//   Device 24 <-> TcCOM Objects/XTS ProcessingUnit 1/Part 1/Module 55
//     Term 109 (AT2002-0250)/CC Inputs/Current actual value Ch.1 <-> Data Pointer/CurrentActualValues[0]
//     Term 109 (AT2002-0250)/CC Inputs/Current actual value Ch.10 <-> Data Pointer/CurrentActualValues[9]
//     Term 109 (AT2002-0250)/CC Inputs/Current actual value Ch.11 <-> Data Pointer/CurrentActualValues[10]
//     Term 109 (AT2002-0250)/CC Inputs/Current actual value Ch.12 <-> Data Pointer/CurrentActualValues[11]
//     Term 109 (AT2002-0250)/CC Inputs/Current actual value Ch.13 <-> Data Pointer/CurrentActualValues[12]
//     Term 109 (AT2002-0250)/CC Inputs/Current actual value Ch.14 <-> Data Pointer/CurrentActualValues[13]
//     Term 109 (AT2002-0250)/CC Inputs/Current actual value Ch.15 <-> Data Pointer/CurrentActualValues[14]
//     Term 109 (AT2002-0250)/CC Inputs/Current actual value Ch.2 <-> Data Pointer/CurrentActualValues[1]
//     Term 109 (AT2002-0250)/CC Inputs/Current actual value Ch.3 <-> Data Pointer/CurrentActualValues[2]
//     Term 109 (AT2002-0250)/CC Inputs/Current actual value Ch.4 <-> Data Pointer/CurrentActualValues[3]
//     Term 109 (AT2002-0250)/CC Inputs/Current actual value Ch.5 <-> Data Pointer/CurrentActualValues[4]
//     Term 109 (AT2002-0250)/CC Inputs/Current actual value Ch.6 <-> Data Pointer/CurrentActualValues[5]
//     Term 109 (AT2002-0250)/CC Inputs/Current actual value Ch.7 <-> Data Pointer/CurrentActualValues[6]
//     Term 109 (AT2002-0250)/CC Inputs/Current actual value Ch.8 <-> Data Pointer/CurrentActualValues[7]
//     Term 109 (AT2002-0250)/CC Inputs/Current actual value Ch.9 <-> Data Pointer/CurrentActualValues[8]
//     Term 109 (AT2002-0250)/CC Inputs/Status <-> Data Pointer/Status
//     Term 109 (AT2002-0250)/CC Outputs/Control <-> Data Pointer/Control
//     Term 109 (AT2002-0250)/CC Outputs/Current setpoint value Ch.1 <-> Data Pointer/CurrentSetpointValues[0]
//     Term 109 (AT2002-0250)/CC Outputs/Current setpoint value Ch.10 <-> Data Pointer/CurrentSetpointValues[9]
//     Term 109 (AT2002-0250)/CC Outputs/Current setpoint value Ch.11 <-> Data Pointer/CurrentSetpointValues[10]
//     Term 109 (AT2002-0250)/CC Outputs/Current setpoint value Ch.12 <-> Data Pointer/CurrentSetpointValues[11]
//     Term 109 (AT2002-0250)/CC Outputs/Current setpoint value Ch.13 <-> Data Pointer/CurrentSetpointValues[12]
//     Term 109 (AT2002-0250)/CC Outputs/Current setpoint value Ch.14 <-> Data Pointer/CurrentSetpointValues[13]
//     Term 109 (AT2002-0250)/CC Outputs/Current setpoint value Ch.15 <-> Data Pointer/CurrentSetpointValues[14]
//     Term 109 (AT2002-0250)/CC Outputs/Current setpoint value Ch.2 <-> Data Pointer/CurrentSetpointValues[1]
//     Term 109 (AT2002-0250)/CC Outputs/Current setpoint value Ch.3 <-> Data Pointer/CurrentSetpointValues[2]
//     Term 109 (AT2002-0250)/CC Outputs/Current setpoint value Ch.4 <-> Data Pointer/CurrentSetpointValues[3]
//     Term 109 (AT2002-0250)/CC Outputs/Current setpoint value Ch.5 <-> Data Pointer/CurrentSetpointValues[4]
//     Term 109 (AT2002-0250)/CC Outputs/Current setpoint value Ch.6 <-> Data Pointer/CurrentSetpointValues[5]
//     Term 109 (AT2002-0250)/CC Outputs/Current setpoint value Ch.7 <-> Data Pointer/CurrentSetpointValues[6]
//     Term 109 (AT2002-0250)/CC Outputs/Current setpoint value Ch.8 <-> Data Pointer/CurrentSetpointValues[7]
//     Term 109 (AT2002-0250)/CC Outputs/Current setpoint value Ch.9 <-> Data Pointer/CurrentSetpointValues[8]
//     Term 109 (AT2002-0250)/Term 110 (AT2002-5250)/FB Inputs/Value Channel 01 <-> Data Pointer/RawPositionValues[0]
//     Term 109 (AT2002-0250)/Term 110 (AT2002-5250)/FB Inputs/Value Channel 02 <-> Data Pointer/RawPositionValues[1]
//     Term 109 (AT2002-0250)/Term 110 (AT2002-5250)/FB Inputs/Value Channel 03 <-> Data Pointer/RawPositionValues[2]
//     Term 109 (AT2002-0250)/Term 110 (AT2002-5250)/FB Inputs/Value Channel 04 <-> Data Pointer/RawPositionValues[3]
//     Term 109 (AT2002-0250)/Term 110 (AT2002-5250)/FB Inputs/Value Channel 05 <-> Data Pointer/RawPositionValues[4]
//     Term 109 (AT2002-0250)/Term 110 (AT2002-5250)/FB Inputs/Value Channel 06 <-> Data Pointer/RawPositionValues[5]
//     Term 109 (AT2002-0250)/Term 110 (AT2002-5250)/FB Inputs/Value Channel 07 <-> Data Pointer/RawPositionValues[6]
//     Term 109 (AT2002-0250)/Term 110 (AT2002-5250)/FB Inputs/Value Channel 08 <-> Data Pointer/RawPositionValues[7]
//     Term 109 (AT2002-0250)/Term 110 (AT2002-5250)/FB Inputs/Value Channel 09 <-> Data Pointer/RawPositionValues[8]
//     Term 109 (AT2002-0250)/Term 110 (AT2002-5250)/FB Inputs/Value Channel 10 <-> Data Pointer/RawPositionValues[9]
//     Term 109 (AT2002-0250)/Term 110 (AT2002-5250)/FB Inputs/Value Channel 11 <-> Data Pointer/RawPositionValues[10]
//     Term 109 (AT2002-0250)/Term 110 (AT2002-5250)/FB Inputs/Value Channel 12 <-> Data Pointer/RawPositionValues[11]
//     Term 109 (AT2002-0250)/Term 110 (AT2002-5250)/FB Inputs/Value Channel 13 <-> Data Pointer/RawPositionValues[12]
//     Term 109 (AT2002-0250)/Term 110 (AT2002-5250)/FB Inputs/Value Channel 14 <-> Data Pointer/RawPositionValues[13]
//     Term 109 (AT2002-0250)/Term 110 (AT2002-5250)/FB Inputs/Value Channel 15 <-> Data Pointer/RawPositionValues[14]
//     Term 109 (AT2002-0250)/Term 110 (AT2002-5250)/FB Inputs/Value Channel 16 <-> Data Pointer/RawPositionValues[15]
//     Term 109 (AT2002-0250)/Term 110 (AT2002-5250)/FB Inputs/Value Channel 17 <-> Data Pointer/RawPositionValues[16]
//     Term 109 (AT2002-0250)/Term 110 (AT2002-5250)/FB Inputs/Value Channel 18 <-> Data Pointer/RawPositionValues[17]
//     Term 109 (AT2002-0250)/Term 110 (AT2002-5250)/FB Inputs/Value Channel 19 <-> Data Pointer/RawPositionValues[18]
//     Term 109 (AT2002-0250)/Term 110 (AT2002-5250)/FB Inputs/Value Channel 20 <-> Data Pointer/RawPositionValues[19]
//     Term 109 (AT2002-0250)/Term 110 (AT2002-5250)/FB Inputs/Value Channel 21 <-> Data Pointer/RawPositionValues[20]
//     Term 109 (AT2002-0250)/Term 110 (AT2002-5250)/FB Inputs/Value Channel 22 <-> Data Pointer/RawPositionValues[21]
//     Term 109 (AT2002-0250)/Term 110 (AT2002-5250)/FB Inputs/Value Channel 23 <-> Data Pointer/RawPositionValues[22]
//     Term 109 (AT2002-0250)/Term 110 (AT2002-5250)/FB Inputs/Value Channel 24 <-> Data Pointer/RawPositionValues[23]
//     Term 109 (AT2002-0250)/Term 110 (AT2002-5250)/FB Inputs/Value Channel 25 <-> Data Pointer/RawPositionValues[24]
//     Term 109 (AT2002-0250)/Term 110 (AT2002-5250)/FB Inputs/Value Channel 26 <-> Data Pointer/RawPositionValues[25]
//     Term 109 (AT2002-0250)/Term 110 (AT2002-5250)/FB Inputs/Value Channel 27 <-> Data Pointer/RawPositionValues[26]
//     Term 109 (AT2002-0250)/Term 110 (AT2002-5250)/FB Inputs/Value Channel 28 <-> Data Pointer/RawPositionValues[27]
//     Term 109 (AT2002-0250)/Term 110 (AT2002-5250)/FB Inputs/Value Channel 29 <-> Data Pointer/RawPositionValues[28]
//     Term 109 (AT2002-0250)/Term 110 (AT2002-5250)/FB Inputs/Value Channel 30 <-> Data Pointer/RawPositionValues[29]
//     Term 109 (AT2002-0250)/Term 110 (AT2002-5250)/FB Inputs/Value Channel 31 <-> Data Pointer/RawPositionValues[30]
//     Term 109 (AT2002-0250)/Term 110 (AT2002-5250)/FB Inputs/Value Channel 32 <-> Data Pointer/RawPositionValues[31]
//   Device 24 <-> TcCOM Objects/XTS ProcessingUnit 1/Part 1/Module 56
//     Term 111 (AT2000-0250)/CC Inputs/Current actual value Ch.1 <-> Data Pointer/CurrentActualValues[0]
//     Term 111 (AT2000-0250)/CC Inputs/Current actual value Ch.10 <-> Data Pointer/CurrentActualValues[9]
//     Term 111 (AT2000-0250)/CC Inputs/Current actual value Ch.11 <-> Data Pointer/CurrentActualValues[10]
//     Term 111 (AT2000-0250)/CC Inputs/Current actual value Ch.12 <-> Data Pointer/CurrentActualValues[11]
//     Term 111 (AT2000-0250)/CC Inputs/Current actual value Ch.13 <-> Data Pointer/CurrentActualValues[12]
//     Term 111 (AT2000-0250)/CC Inputs/Current actual value Ch.14 <-> Data Pointer/CurrentActualValues[13]
//     Term 111 (AT2000-0250)/CC Inputs/Current actual value Ch.15 <-> Data Pointer/CurrentActualValues[14]
//     Term 111 (AT2000-0250)/CC Inputs/Current actual value Ch.2 <-> Data Pointer/CurrentActualValues[1]
//     Term 111 (AT2000-0250)/CC Inputs/Current actual value Ch.3 <-> Data Pointer/CurrentActualValues[2]
//     Term 111 (AT2000-0250)/CC Inputs/Current actual value Ch.4 <-> Data Pointer/CurrentActualValues[3]
//     Term 111 (AT2000-0250)/CC Inputs/Current actual value Ch.5 <-> Data Pointer/CurrentActualValues[4]
//     Term 111 (AT2000-0250)/CC Inputs/Current actual value Ch.6 <-> Data Pointer/CurrentActualValues[5]
//     Term 111 (AT2000-0250)/CC Inputs/Current actual value Ch.7 <-> Data Pointer/CurrentActualValues[6]
//     Term 111 (AT2000-0250)/CC Inputs/Current actual value Ch.8 <-> Data Pointer/CurrentActualValues[7]
//     Term 111 (AT2000-0250)/CC Inputs/Current actual value Ch.9 <-> Data Pointer/CurrentActualValues[8]
//     Term 111 (AT2000-0250)/CC Inputs/Status <-> Data Pointer/Status
//     Term 111 (AT2000-0250)/CC Outputs/Control <-> Data Pointer/Control
//     Term 111 (AT2000-0250)/CC Outputs/Current setpoint value Ch.1 <-> Data Pointer/CurrentSetpointValues[0]
//     Term 111 (AT2000-0250)/CC Outputs/Current setpoint value Ch.10 <-> Data Pointer/CurrentSetpointValues[9]
//     Term 111 (AT2000-0250)/CC Outputs/Current setpoint value Ch.11 <-> Data Pointer/CurrentSetpointValues[10]
//     Term 111 (AT2000-0250)/CC Outputs/Current setpoint value Ch.12 <-> Data Pointer/CurrentSetpointValues[11]
//     Term 111 (AT2000-0250)/CC Outputs/Current setpoint value Ch.13 <-> Data Pointer/CurrentSetpointValues[12]
//     Term 111 (AT2000-0250)/CC Outputs/Current setpoint value Ch.14 <-> Data Pointer/CurrentSetpointValues[13]
//     Term 111 (AT2000-0250)/CC Outputs/Current setpoint value Ch.15 <-> Data Pointer/CurrentSetpointValues[14]
//     Term 111 (AT2000-0250)/CC Outputs/Current setpoint value Ch.2 <-> Data Pointer/CurrentSetpointValues[1]
//     Term 111 (AT2000-0250)/CC Outputs/Current setpoint value Ch.3 <-> Data Pointer/CurrentSetpointValues[2]
//     Term 111 (AT2000-0250)/CC Outputs/Current setpoint value Ch.4 <-> Data Pointer/CurrentSetpointValues[3]
//     Term 111 (AT2000-0250)/CC Outputs/Current setpoint value Ch.5 <-> Data Pointer/CurrentSetpointValues[4]
//     Term 111 (AT2000-0250)/CC Outputs/Current setpoint value Ch.6 <-> Data Pointer/CurrentSetpointValues[5]
//     Term 111 (AT2000-0250)/CC Outputs/Current setpoint value Ch.7 <-> Data Pointer/CurrentSetpointValues[6]
//     Term 111 (AT2000-0250)/CC Outputs/Current setpoint value Ch.8 <-> Data Pointer/CurrentSetpointValues[7]
//     Term 111 (AT2000-0250)/CC Outputs/Current setpoint value Ch.9 <-> Data Pointer/CurrentSetpointValues[8]
//     Term 111 (AT2000-0250)/Term 112 (AT2000-5250)/FB Inputs/Value Channel 01 <-> Data Pointer/RawPositionValues[0]
//     Term 111 (AT2000-0250)/Term 112 (AT2000-5250)/FB Inputs/Value Channel 02 <-> Data Pointer/RawPositionValues[1]
//     Term 111 (AT2000-0250)/Term 112 (AT2000-5250)/FB Inputs/Value Channel 03 <-> Data Pointer/RawPositionValues[2]
//     Term 111 (AT2000-0250)/Term 112 (AT2000-5250)/FB Inputs/Value Channel 04 <-> Data Pointer/RawPositionValues[3]
//     Term 111 (AT2000-0250)/Term 112 (AT2000-5250)/FB Inputs/Value Channel 05 <-> Data Pointer/RawPositionValues[4]
//     Term 111 (AT2000-0250)/Term 112 (AT2000-5250)/FB Inputs/Value Channel 06 <-> Data Pointer/RawPositionValues[5]
//     Term 111 (AT2000-0250)/Term 112 (AT2000-5250)/FB Inputs/Value Channel 07 <-> Data Pointer/RawPositionValues[6]
//     Term 111 (AT2000-0250)/Term 112 (AT2000-5250)/FB Inputs/Value Channel 08 <-> Data Pointer/RawPositionValues[7]
//     Term 111 (AT2000-0250)/Term 112 (AT2000-5250)/FB Inputs/Value Channel 09 <-> Data Pointer/RawPositionValues[8]
//     Term 111 (AT2000-0250)/Term 112 (AT2000-5250)/FB Inputs/Value Channel 10 <-> Data Pointer/RawPositionValues[9]
//     Term 111 (AT2000-0250)/Term 112 (AT2000-5250)/FB Inputs/Value Channel 11 <-> Data Pointer/RawPositionValues[10]
//     Term 111 (AT2000-0250)/Term 112 (AT2000-5250)/FB Inputs/Value Channel 12 <-> Data Pointer/RawPositionValues[11]
//     Term 111 (AT2000-0250)/Term 112 (AT2000-5250)/FB Inputs/Value Channel 13 <-> Data Pointer/RawPositionValues[12]
//     Term 111 (AT2000-0250)/Term 112 (AT2000-5250)/FB Inputs/Value Channel 14 <-> Data Pointer/RawPositionValues[13]
//     Term 111 (AT2000-0250)/Term 112 (AT2000-5250)/FB Inputs/Value Channel 15 <-> Data Pointer/RawPositionValues[14]
//     Term 111 (AT2000-0250)/Term 112 (AT2000-5250)/FB Inputs/Value Channel 16 <-> Data Pointer/RawPositionValues[15]
//     Term 111 (AT2000-0250)/Term 112 (AT2000-5250)/FB Inputs/Value Channel 17 <-> Data Pointer/RawPositionValues[16]
//     Term 111 (AT2000-0250)/Term 112 (AT2000-5250)/FB Inputs/Value Channel 18 <-> Data Pointer/RawPositionValues[17]
//     Term 111 (AT2000-0250)/Term 112 (AT2000-5250)/FB Inputs/Value Channel 19 <-> Data Pointer/RawPositionValues[18]
//     Term 111 (AT2000-0250)/Term 112 (AT2000-5250)/FB Inputs/Value Channel 20 <-> Data Pointer/RawPositionValues[19]
//     Term 111 (AT2000-0250)/Term 112 (AT2000-5250)/FB Inputs/Value Channel 21 <-> Data Pointer/RawPositionValues[20]
//     Term 111 (AT2000-0250)/Term 112 (AT2000-5250)/FB Inputs/Value Channel 22 <-> Data Pointer/RawPositionValues[21]
//     Term 111 (AT2000-0250)/Term 112 (AT2000-5250)/FB Inputs/Value Channel 23 <-> Data Pointer/RawPositionValues[22]
//     Term 111 (AT2000-0250)/Term 112 (AT2000-5250)/FB Inputs/Value Channel 24 <-> Data Pointer/RawPositionValues[23]
//     Term 111 (AT2000-0250)/Term 112 (AT2000-5250)/FB Inputs/Value Channel 25 <-> Data Pointer/RawPositionValues[24]
//     Term 111 (AT2000-0250)/Term 112 (AT2000-5250)/FB Inputs/Value Channel 26 <-> Data Pointer/RawPositionValues[25]
//     Term 111 (AT2000-0250)/Term 112 (AT2000-5250)/FB Inputs/Value Channel 27 <-> Data Pointer/RawPositionValues[26]
//     Term 111 (AT2000-0250)/Term 112 (AT2000-5250)/FB Inputs/Value Channel 28 <-> Data Pointer/RawPositionValues[27]
//     Term 111 (AT2000-0250)/Term 112 (AT2000-5250)/FB Inputs/Value Channel 29 <-> Data Pointer/RawPositionValues[28]
//     Term 111 (AT2000-0250)/Term 112 (AT2000-5250)/FB Inputs/Value Channel 30 <-> Data Pointer/RawPositionValues[29]
//     Term 111 (AT2000-0250)/Term 112 (AT2000-5250)/FB Inputs/Value Channel 31 <-> Data Pointer/RawPositionValues[30]
//     Term 111 (AT2000-0250)/Term 112 (AT2000-5250)/FB Inputs/Value Channel 32 <-> Data Pointer/RawPositionValues[31]
//   Device 24 <-> TcCOM Objects/XTS ProcessingUnit 1/Part 1/Module 57
//     Term 113 (AT2000-0250)/CC Inputs/Current actual value Ch.1 <-> Data Pointer/CurrentActualValues[0]
//     Term 113 (AT2000-0250)/CC Inputs/Current actual value Ch.10 <-> Data Pointer/CurrentActualValues[9]
//     Term 113 (AT2000-0250)/CC Inputs/Current actual value Ch.11 <-> Data Pointer/CurrentActualValues[10]
//     Term 113 (AT2000-0250)/CC Inputs/Current actual value Ch.12 <-> Data Pointer/CurrentActualValues[11]
//     Term 113 (AT2000-0250)/CC Inputs/Current actual value Ch.13 <-> Data Pointer/CurrentActualValues[12]
//     Term 113 (AT2000-0250)/CC Inputs/Current actual value Ch.14 <-> Data Pointer/CurrentActualValues[13]
//     Term 113 (AT2000-0250)/CC Inputs/Current actual value Ch.15 <-> Data Pointer/CurrentActualValues[14]
//     Term 113 (AT2000-0250)/CC Inputs/Current actual value Ch.2 <-> Data Pointer/CurrentActualValues[1]
//     Term 113 (AT2000-0250)/CC Inputs/Current actual value Ch.3 <-> Data Pointer/CurrentActualValues[2]
//     Term 113 (AT2000-0250)/CC Inputs/Current actual value Ch.4 <-> Data Pointer/CurrentActualValues[3]
//     Term 113 (AT2000-0250)/CC Inputs/Current actual value Ch.5 <-> Data Pointer/CurrentActualValues[4]
//     Term 113 (AT2000-0250)/CC Inputs/Current actual value Ch.6 <-> Data Pointer/CurrentActualValues[5]
//     Term 113 (AT2000-0250)/CC Inputs/Current actual value Ch.7 <-> Data Pointer/CurrentActualValues[6]
//     Term 113 (AT2000-0250)/CC Inputs/Current actual value Ch.8 <-> Data Pointer/CurrentActualValues[7]
//     Term 113 (AT2000-0250)/CC Inputs/Current actual value Ch.9 <-> Data Pointer/CurrentActualValues[8]
//     Term 113 (AT2000-0250)/CC Inputs/Status <-> Data Pointer/Status
//     Term 113 (AT2000-0250)/CC Outputs/Control <-> Data Pointer/Control
//     Term 113 (AT2000-0250)/CC Outputs/Current setpoint value Ch.1 <-> Data Pointer/CurrentSetpointValues[0]
//     Term 113 (AT2000-0250)/CC Outputs/Current setpoint value Ch.10 <-> Data Pointer/CurrentSetpointValues[9]
//     Term 113 (AT2000-0250)/CC Outputs/Current setpoint value Ch.11 <-> Data Pointer/CurrentSetpointValues[10]
//     Term 113 (AT2000-0250)/CC Outputs/Current setpoint value Ch.12 <-> Data Pointer/CurrentSetpointValues[11]
//     Term 113 (AT2000-0250)/CC Outputs/Current setpoint value Ch.13 <-> Data Pointer/CurrentSetpointValues[12]
//     Term 113 (AT2000-0250)/CC Outputs/Current setpoint value Ch.14 <-> Data Pointer/CurrentSetpointValues[13]
//     Term 113 (AT2000-0250)/CC Outputs/Current setpoint value Ch.15 <-> Data Pointer/CurrentSetpointValues[14]
//     Term 113 (AT2000-0250)/CC Outputs/Current setpoint value Ch.2 <-> Data Pointer/CurrentSetpointValues[1]
//     Term 113 (AT2000-0250)/CC Outputs/Current setpoint value Ch.3 <-> Data Pointer/CurrentSetpointValues[2]
//     Term 113 (AT2000-0250)/CC Outputs/Current setpoint value Ch.4 <-> Data Pointer/CurrentSetpointValues[3]
//     Term 113 (AT2000-0250)/CC Outputs/Current setpoint value Ch.5 <-> Data Pointer/CurrentSetpointValues[4]
//     Term 113 (AT2000-0250)/CC Outputs/Current setpoint value Ch.6 <-> Data Pointer/CurrentSetpointValues[5]
//     Term 113 (AT2000-0250)/CC Outputs/Current setpoint value Ch.7 <-> Data Pointer/CurrentSetpointValues[6]
//     Term 113 (AT2000-0250)/CC Outputs/Current setpoint value Ch.8 <-> Data Pointer/CurrentSetpointValues[7]
//     Term 113 (AT2000-0250)/CC Outputs/Current setpoint value Ch.9 <-> Data Pointer/CurrentSetpointValues[8]
//     Term 113 (AT2000-0250)/Term 114 (AT2000-5250)/FB Inputs/Value Channel 01 <-> Data Pointer/RawPositionValues[0]
//     Term 113 (AT2000-0250)/Term 114 (AT2000-5250)/FB Inputs/Value Channel 02 <-> Data Pointer/RawPositionValues[1]
//     Term 113 (AT2000-0250)/Term 114 (AT2000-5250)/FB Inputs/Value Channel 03 <-> Data Pointer/RawPositionValues[2]
//     Term 113 (AT2000-0250)/Term 114 (AT2000-5250)/FB Inputs/Value Channel 04 <-> Data Pointer/RawPositionValues[3]
//     Term 113 (AT2000-0250)/Term 114 (AT2000-5250)/FB Inputs/Value Channel 05 <-> Data Pointer/RawPositionValues[4]
//     Term 113 (AT2000-0250)/Term 114 (AT2000-5250)/FB Inputs/Value Channel 06 <-> Data Pointer/RawPositionValues[5]
//     Term 113 (AT2000-0250)/Term 114 (AT2000-5250)/FB Inputs/Value Channel 07 <-> Data Pointer/RawPositionValues[6]
//     Term 113 (AT2000-0250)/Term 114 (AT2000-5250)/FB Inputs/Value Channel 08 <-> Data Pointer/RawPositionValues[7]
//     Term 113 (AT2000-0250)/Term 114 (AT2000-5250)/FB Inputs/Value Channel 09 <-> Data Pointer/RawPositionValues[8]
//     Term 113 (AT2000-0250)/Term 114 (AT2000-5250)/FB Inputs/Value Channel 10 <-> Data Pointer/RawPositionValues[9]
//     Term 113 (AT2000-0250)/Term 114 (AT2000-5250)/FB Inputs/Value Channel 11 <-> Data Pointer/RawPositionValues[10]
//     Term 113 (AT2000-0250)/Term 114 (AT2000-5250)/FB Inputs/Value Channel 12 <-> Data Pointer/RawPositionValues[11]
//     Term 113 (AT2000-0250)/Term 114 (AT2000-5250)/FB Inputs/Value Channel 13 <-> Data Pointer/RawPositionValues[12]
//     Term 113 (AT2000-0250)/Term 114 (AT2000-5250)/FB Inputs/Value Channel 14 <-> Data Pointer/RawPositionValues[13]
//     Term 113 (AT2000-0250)/Term 114 (AT2000-5250)/FB Inputs/Value Channel 15 <-> Data Pointer/RawPositionValues[14]
//     Term 113 (AT2000-0250)/Term 114 (AT2000-5250)/FB Inputs/Value Channel 16 <-> Data Pointer/RawPositionValues[15]
//     Term 113 (AT2000-0250)/Term 114 (AT2000-5250)/FB Inputs/Value Channel 17 <-> Data Pointer/RawPositionValues[16]
//     Term 113 (AT2000-0250)/Term 114 (AT2000-5250)/FB Inputs/Value Channel 18 <-> Data Pointer/RawPositionValues[17]
//     Term 113 (AT2000-0250)/Term 114 (AT2000-5250)/FB Inputs/Value Channel 19 <-> Data Pointer/RawPositionValues[18]
//     Term 113 (AT2000-0250)/Term 114 (AT2000-5250)/FB Inputs/Value Channel 20 <-> Data Pointer/RawPositionValues[19]
//     Term 113 (AT2000-0250)/Term 114 (AT2000-5250)/FB Inputs/Value Channel 21 <-> Data Pointer/RawPositionValues[20]
//     Term 113 (AT2000-0250)/Term 114 (AT2000-5250)/FB Inputs/Value Channel 22 <-> Data Pointer/RawPositionValues[21]
//     Term 113 (AT2000-0250)/Term 114 (AT2000-5250)/FB Inputs/Value Channel 23 <-> Data Pointer/RawPositionValues[22]
//     Term 113 (AT2000-0250)/Term 114 (AT2000-5250)/FB Inputs/Value Channel 24 <-> Data Pointer/RawPositionValues[23]
//     Term 113 (AT2000-0250)/Term 114 (AT2000-5250)/FB Inputs/Value Channel 25 <-> Data Pointer/RawPositionValues[24]
//     Term 113 (AT2000-0250)/Term 114 (AT2000-5250)/FB Inputs/Value Channel 26 <-> Data Pointer/RawPositionValues[25]
//     Term 113 (AT2000-0250)/Term 114 (AT2000-5250)/FB Inputs/Value Channel 27 <-> Data Pointer/RawPositionValues[26]
//     Term 113 (AT2000-0250)/Term 114 (AT2000-5250)/FB Inputs/Value Channel 28 <-> Data Pointer/RawPositionValues[27]
//     Term 113 (AT2000-0250)/Term 114 (AT2000-5250)/FB Inputs/Value Channel 29 <-> Data Pointer/RawPositionValues[28]
//     Term 113 (AT2000-0250)/Term 114 (AT2000-5250)/FB Inputs/Value Channel 30 <-> Data Pointer/RawPositionValues[29]
//     Term 113 (AT2000-0250)/Term 114 (AT2000-5250)/FB Inputs/Value Channel 31 <-> Data Pointer/RawPositionValues[30]
//     Term 113 (AT2000-0250)/Term 114 (AT2000-5250)/FB Inputs/Value Channel 32 <-> Data Pointer/RawPositionValues[31]
//   Device 24 <-> TcCOM Objects/XTS ProcessingUnit 1/Part 1/Module 58
//     Term 115 (AT2000-0250)/CC Inputs/Current actual value Ch.1 <-> Data Pointer/CurrentActualValues[0]
//     Term 115 (AT2000-0250)/CC Inputs/Current actual value Ch.10 <-> Data Pointer/CurrentActualValues[9]
//     Term 115 (AT2000-0250)/CC Inputs/Current actual value Ch.11 <-> Data Pointer/CurrentActualValues[10]
//     Term 115 (AT2000-0250)/CC Inputs/Current actual value Ch.12 <-> Data Pointer/CurrentActualValues[11]
//     Term 115 (AT2000-0250)/CC Inputs/Current actual value Ch.13 <-> Data Pointer/CurrentActualValues[12]
//     Term 115 (AT2000-0250)/CC Inputs/Current actual value Ch.14 <-> Data Pointer/CurrentActualValues[13]
//     Term 115 (AT2000-0250)/CC Inputs/Current actual value Ch.15 <-> Data Pointer/CurrentActualValues[14]
//     Term 115 (AT2000-0250)/CC Inputs/Current actual value Ch.2 <-> Data Pointer/CurrentActualValues[1]
//     Term 115 (AT2000-0250)/CC Inputs/Current actual value Ch.3 <-> Data Pointer/CurrentActualValues[2]
//     Term 115 (AT2000-0250)/CC Inputs/Current actual value Ch.4 <-> Data Pointer/CurrentActualValues[3]
//     Term 115 (AT2000-0250)/CC Inputs/Current actual value Ch.5 <-> Data Pointer/CurrentActualValues[4]
//     Term 115 (AT2000-0250)/CC Inputs/Current actual value Ch.6 <-> Data Pointer/CurrentActualValues[5]
//     Term 115 (AT2000-0250)/CC Inputs/Current actual value Ch.7 <-> Data Pointer/CurrentActualValues[6]
//     Term 115 (AT2000-0250)/CC Inputs/Current actual value Ch.8 <-> Data Pointer/CurrentActualValues[7]
//     Term 115 (AT2000-0250)/CC Inputs/Current actual value Ch.9 <-> Data Pointer/CurrentActualValues[8]
//     Term 115 (AT2000-0250)/CC Inputs/Status <-> Data Pointer/Status
//     Term 115 (AT2000-0250)/CC Outputs/Control <-> Data Pointer/Control
//     Term 115 (AT2000-0250)/CC Outputs/Current setpoint value Ch.1 <-> Data Pointer/CurrentSetpointValues[0]
//     Term 115 (AT2000-0250)/CC Outputs/Current setpoint value Ch.10 <-> Data Pointer/CurrentSetpointValues[9]
//     Term 115 (AT2000-0250)/CC Outputs/Current setpoint value Ch.11 <-> Data Pointer/CurrentSetpointValues[10]
//     Term 115 (AT2000-0250)/CC Outputs/Current setpoint value Ch.12 <-> Data Pointer/CurrentSetpointValues[11]
//     Term 115 (AT2000-0250)/CC Outputs/Current setpoint value Ch.13 <-> Data Pointer/CurrentSetpointValues[12]
//     Term 115 (AT2000-0250)/CC Outputs/Current setpoint value Ch.14 <-> Data Pointer/CurrentSetpointValues[13]
//     Term 115 (AT2000-0250)/CC Outputs/Current setpoint value Ch.15 <-> Data Pointer/CurrentSetpointValues[14]
//     Term 115 (AT2000-0250)/CC Outputs/Current setpoint value Ch.2 <-> Data Pointer/CurrentSetpointValues[1]
//     Term 115 (AT2000-0250)/CC Outputs/Current setpoint value Ch.3 <-> Data Pointer/CurrentSetpointValues[2]
//     Term 115 (AT2000-0250)/CC Outputs/Current setpoint value Ch.4 <-> Data Pointer/CurrentSetpointValues[3]
//     Term 115 (AT2000-0250)/CC Outputs/Current setpoint value Ch.5 <-> Data Pointer/CurrentSetpointValues[4]
//     Term 115 (AT2000-0250)/CC Outputs/Current setpoint value Ch.6 <-> Data Pointer/CurrentSetpointValues[5]
//     Term 115 (AT2000-0250)/CC Outputs/Current setpoint value Ch.7 <-> Data Pointer/CurrentSetpointValues[6]
//     Term 115 (AT2000-0250)/CC Outputs/Current setpoint value Ch.8 <-> Data Pointer/CurrentSetpointValues[7]
//     Term 115 (AT2000-0250)/CC Outputs/Current setpoint value Ch.9 <-> Data Pointer/CurrentSetpointValues[8]
//     Term 115 (AT2000-0250)/Term 116 (AT2000-5250)/FB Inputs/Value Channel 01 <-> Data Pointer/RawPositionValues[0]
//     Term 115 (AT2000-0250)/Term 116 (AT2000-5250)/FB Inputs/Value Channel 02 <-> Data Pointer/RawPositionValues[1]
//     Term 115 (AT2000-0250)/Term 116 (AT2000-5250)/FB Inputs/Value Channel 03 <-> Data Pointer/RawPositionValues[2]
//     Term 115 (AT2000-0250)/Term 116 (AT2000-5250)/FB Inputs/Value Channel 04 <-> Data Pointer/RawPositionValues[3]
//     Term 115 (AT2000-0250)/Term 116 (AT2000-5250)/FB Inputs/Value Channel 05 <-> Data Pointer/RawPositionValues[4]
//     Term 115 (AT2000-0250)/Term 116 (AT2000-5250)/FB Inputs/Value Channel 06 <-> Data Pointer/RawPositionValues[5]
//     Term 115 (AT2000-0250)/Term 116 (AT2000-5250)/FB Inputs/Value Channel 07 <-> Data Pointer/RawPositionValues[6]
//     Term 115 (AT2000-0250)/Term 116 (AT2000-5250)/FB Inputs/Value Channel 08 <-> Data Pointer/RawPositionValues[7]
//     Term 115 (AT2000-0250)/Term 116 (AT2000-5250)/FB Inputs/Value Channel 09 <-> Data Pointer/RawPositionValues[8]
//     Term 115 (AT2000-0250)/Term 116 (AT2000-5250)/FB Inputs/Value Channel 10 <-> Data Pointer/RawPositionValues[9]
//     Term 115 (AT2000-0250)/Term 116 (AT2000-5250)/FB Inputs/Value Channel 11 <-> Data Pointer/RawPositionValues[10]
//     Term 115 (AT2000-0250)/Term 116 (AT2000-5250)/FB Inputs/Value Channel 12 <-> Data Pointer/RawPositionValues[11]
//     Term 115 (AT2000-0250)/Term 116 (AT2000-5250)/FB Inputs/Value Channel 13 <-> Data Pointer/RawPositionValues[12]
//     Term 115 (AT2000-0250)/Term 116 (AT2000-5250)/FB Inputs/Value Channel 14 <-> Data Pointer/RawPositionValues[13]
//     Term 115 (AT2000-0250)/Term 116 (AT2000-5250)/FB Inputs/Value Channel 15 <-> Data Pointer/RawPositionValues[14]
//     Term 115 (AT2000-0250)/Term 116 (AT2000-5250)/FB Inputs/Value Channel 16 <-> Data Pointer/RawPositionValues[15]
//     Term 115 (AT2000-0250)/Term 116 (AT2000-5250)/FB Inputs/Value Channel 17 <-> Data Pointer/RawPositionValues[16]
//     Term 115 (AT2000-0250)/Term 116 (AT2000-5250)/FB Inputs/Value Channel 18 <-> Data Pointer/RawPositionValues[17]
//     Term 115 (AT2000-0250)/Term 116 (AT2000-5250)/FB Inputs/Value Channel 19 <-> Data Pointer/RawPositionValues[18]
//     Term 115 (AT2000-0250)/Term 116 (AT2000-5250)/FB Inputs/Value Channel 20 <-> Data Pointer/RawPositionValues[19]
//     Term 115 (AT2000-0250)/Term 116 (AT2000-5250)/FB Inputs/Value Channel 21 <-> Data Pointer/RawPositionValues[20]
//     Term 115 (AT2000-0250)/Term 116 (AT2000-5250)/FB Inputs/Value Channel 22 <-> Data Pointer/RawPositionValues[21]
//     Term 115 (AT2000-0250)/Term 116 (AT2000-5250)/FB Inputs/Value Channel 23 <-> Data Pointer/RawPositionValues[22]
//     Term 115 (AT2000-0250)/Term 116 (AT2000-5250)/FB Inputs/Value Channel 24 <-> Data Pointer/RawPositionValues[23]
//     Term 115 (AT2000-0250)/Term 116 (AT2000-5250)/FB Inputs/Value Channel 25 <-> Data Pointer/RawPositionValues[24]
//     Term 115 (AT2000-0250)/Term 116 (AT2000-5250)/FB Inputs/Value Channel 26 <-> Data Pointer/RawPositionValues[25]
//     Term 115 (AT2000-0250)/Term 116 (AT2000-5250)/FB Inputs/Value Channel 27 <-> Data Pointer/RawPositionValues[26]
//     Term 115 (AT2000-0250)/Term 116 (AT2000-5250)/FB Inputs/Value Channel 28 <-> Data Pointer/RawPositionValues[27]
//     Term 115 (AT2000-0250)/Term 116 (AT2000-5250)/FB Inputs/Value Channel 29 <-> Data Pointer/RawPositionValues[28]
//     Term 115 (AT2000-0250)/Term 116 (AT2000-5250)/FB Inputs/Value Channel 30 <-> Data Pointer/RawPositionValues[29]
//     Term 115 (AT2000-0250)/Term 116 (AT2000-5250)/FB Inputs/Value Channel 31 <-> Data Pointer/RawPositionValues[30]
//     Term 115 (AT2000-0250)/Term 116 (AT2000-5250)/FB Inputs/Value Channel 32 <-> Data Pointer/RawPositionValues[31]
//   Device 24 <-> TcCOM Objects/XTS ProcessingUnit 1/Part 1/Module 59
//     Term 117 (AT2000-0250)/CC Inputs/Current actual value Ch.1 <-> Data Pointer/CurrentActualValues[0]
//     Term 117 (AT2000-0250)/CC Inputs/Current actual value Ch.10 <-> Data Pointer/CurrentActualValues[9]
//     Term 117 (AT2000-0250)/CC Inputs/Current actual value Ch.11 <-> Data Pointer/CurrentActualValues[10]
//     Term 117 (AT2000-0250)/CC Inputs/Current actual value Ch.12 <-> Data Pointer/CurrentActualValues[11]
//     Term 117 (AT2000-0250)/CC Inputs/Current actual value Ch.13 <-> Data Pointer/CurrentActualValues[12]
//     Term 117 (AT2000-0250)/CC Inputs/Current actual value Ch.14 <-> Data Pointer/CurrentActualValues[13]
//     Term 117 (AT2000-0250)/CC Inputs/Current actual value Ch.15 <-> Data Pointer/CurrentActualValues[14]
//     Term 117 (AT2000-0250)/CC Inputs/Current actual value Ch.2 <-> Data Pointer/CurrentActualValues[1]
//     Term 117 (AT2000-0250)/CC Inputs/Current actual value Ch.3 <-> Data Pointer/CurrentActualValues[2]
//     Term 117 (AT2000-0250)/CC Inputs/Current actual value Ch.4 <-> Data Pointer/CurrentActualValues[3]
//     Term 117 (AT2000-0250)/CC Inputs/Current actual value Ch.5 <-> Data Pointer/CurrentActualValues[4]
//     Term 117 (AT2000-0250)/CC Inputs/Current actual value Ch.6 <-> Data Pointer/CurrentActualValues[5]
//     Term 117 (AT2000-0250)/CC Inputs/Current actual value Ch.7 <-> Data Pointer/CurrentActualValues[6]
//     Term 117 (AT2000-0250)/CC Inputs/Current actual value Ch.8 <-> Data Pointer/CurrentActualValues[7]
//     Term 117 (AT2000-0250)/CC Inputs/Current actual value Ch.9 <-> Data Pointer/CurrentActualValues[8]
//     Term 117 (AT2000-0250)/CC Inputs/Status <-> Data Pointer/Status
//     Term 117 (AT2000-0250)/CC Outputs/Control <-> Data Pointer/Control
//     Term 117 (AT2000-0250)/CC Outputs/Current setpoint value Ch.1 <-> Data Pointer/CurrentSetpointValues[0]
//     Term 117 (AT2000-0250)/CC Outputs/Current setpoint value Ch.10 <-> Data Pointer/CurrentSetpointValues[9]
//     Term 117 (AT2000-0250)/CC Outputs/Current setpoint value Ch.11 <-> Data Pointer/CurrentSetpointValues[10]
//     Term 117 (AT2000-0250)/CC Outputs/Current setpoint value Ch.12 <-> Data Pointer/CurrentSetpointValues[11]
//     Term 117 (AT2000-0250)/CC Outputs/Current setpoint value Ch.13 <-> Data Pointer/CurrentSetpointValues[12]
//     Term 117 (AT2000-0250)/CC Outputs/Current setpoint value Ch.14 <-> Data Pointer/CurrentSetpointValues[13]
//     Term 117 (AT2000-0250)/CC Outputs/Current setpoint value Ch.15 <-> Data Pointer/CurrentSetpointValues[14]
//     Term 117 (AT2000-0250)/CC Outputs/Current setpoint value Ch.2 <-> Data Pointer/CurrentSetpointValues[1]
//     Term 117 (AT2000-0250)/CC Outputs/Current setpoint value Ch.3 <-> Data Pointer/CurrentSetpointValues[2]
//     Term 117 (AT2000-0250)/CC Outputs/Current setpoint value Ch.4 <-> Data Pointer/CurrentSetpointValues[3]
//     Term 117 (AT2000-0250)/CC Outputs/Current setpoint value Ch.5 <-> Data Pointer/CurrentSetpointValues[4]
//     Term 117 (AT2000-0250)/CC Outputs/Current setpoint value Ch.6 <-> Data Pointer/CurrentSetpointValues[5]
//     Term 117 (AT2000-0250)/CC Outputs/Current setpoint value Ch.7 <-> Data Pointer/CurrentSetpointValues[6]
//     Term 117 (AT2000-0250)/CC Outputs/Current setpoint value Ch.8 <-> Data Pointer/CurrentSetpointValues[7]
//     Term 117 (AT2000-0250)/CC Outputs/Current setpoint value Ch.9 <-> Data Pointer/CurrentSetpointValues[8]
//     Term 117 (AT2000-0250)/Term 118 (AT2000-5250)/FB Inputs/Value Channel 01 <-> Data Pointer/RawPositionValues[0]
//     Term 117 (AT2000-0250)/Term 118 (AT2000-5250)/FB Inputs/Value Channel 02 <-> Data Pointer/RawPositionValues[1]
//     Term 117 (AT2000-0250)/Term 118 (AT2000-5250)/FB Inputs/Value Channel 03 <-> Data Pointer/RawPositionValues[2]
//     Term 117 (AT2000-0250)/Term 118 (AT2000-5250)/FB Inputs/Value Channel 04 <-> Data Pointer/RawPositionValues[3]
//     Term 117 (AT2000-0250)/Term 118 (AT2000-5250)/FB Inputs/Value Channel 05 <-> Data Pointer/RawPositionValues[4]
//     Term 117 (AT2000-0250)/Term 118 (AT2000-5250)/FB Inputs/Value Channel 06 <-> Data Pointer/RawPositionValues[5]
//     Term 117 (AT2000-0250)/Term 118 (AT2000-5250)/FB Inputs/Value Channel 07 <-> Data Pointer/RawPositionValues[6]
//     Term 117 (AT2000-0250)/Term 118 (AT2000-5250)/FB Inputs/Value Channel 08 <-> Data Pointer/RawPositionValues[7]
//     Term 117 (AT2000-0250)/Term 118 (AT2000-5250)/FB Inputs/Value Channel 09 <-> Data Pointer/RawPositionValues[8]
//     Term 117 (AT2000-0250)/Term 118 (AT2000-5250)/FB Inputs/Value Channel 10 <-> Data Pointer/RawPositionValues[9]
//     Term 117 (AT2000-0250)/Term 118 (AT2000-5250)/FB Inputs/Value Channel 11 <-> Data Pointer/RawPositionValues[10]
//     Term 117 (AT2000-0250)/Term 118 (AT2000-5250)/FB Inputs/Value Channel 12 <-> Data Pointer/RawPositionValues[11]
//     Term 117 (AT2000-0250)/Term 118 (AT2000-5250)/FB Inputs/Value Channel 13 <-> Data Pointer/RawPositionValues[12]
//     Term 117 (AT2000-0250)/Term 118 (AT2000-5250)/FB Inputs/Value Channel 14 <-> Data Pointer/RawPositionValues[13]
//     Term 117 (AT2000-0250)/Term 118 (AT2000-5250)/FB Inputs/Value Channel 15 <-> Data Pointer/RawPositionValues[14]
//     Term 117 (AT2000-0250)/Term 118 (AT2000-5250)/FB Inputs/Value Channel 16 <-> Data Pointer/RawPositionValues[15]
//     Term 117 (AT2000-0250)/Term 118 (AT2000-5250)/FB Inputs/Value Channel 17 <-> Data Pointer/RawPositionValues[16]
//     Term 117 (AT2000-0250)/Term 118 (AT2000-5250)/FB Inputs/Value Channel 18 <-> Data Pointer/RawPositionValues[17]
//     Term 117 (AT2000-0250)/Term 118 (AT2000-5250)/FB Inputs/Value Channel 19 <-> Data Pointer/RawPositionValues[18]
//     Term 117 (AT2000-0250)/Term 118 (AT2000-5250)/FB Inputs/Value Channel 20 <-> Data Pointer/RawPositionValues[19]
//     Term 117 (AT2000-0250)/Term 118 (AT2000-5250)/FB Inputs/Value Channel 21 <-> Data Pointer/RawPositionValues[20]
//     Term 117 (AT2000-0250)/Term 118 (AT2000-5250)/FB Inputs/Value Channel 22 <-> Data Pointer/RawPositionValues[21]
//     Term 117 (AT2000-0250)/Term 118 (AT2000-5250)/FB Inputs/Value Channel 23 <-> Data Pointer/RawPositionValues[22]
//     Term 117 (AT2000-0250)/Term 118 (AT2000-5250)/FB Inputs/Value Channel 24 <-> Data Pointer/RawPositionValues[23]
//     Term 117 (AT2000-0250)/Term 118 (AT2000-5250)/FB Inputs/Value Channel 25 <-> Data Pointer/RawPositionValues[24]
//     Term 117 (AT2000-0250)/Term 118 (AT2000-5250)/FB Inputs/Value Channel 26 <-> Data Pointer/RawPositionValues[25]
//     Term 117 (AT2000-0250)/Term 118 (AT2000-5250)/FB Inputs/Value Channel 27 <-> Data Pointer/RawPositionValues[26]
//     Term 117 (AT2000-0250)/Term 118 (AT2000-5250)/FB Inputs/Value Channel 28 <-> Data Pointer/RawPositionValues[27]
//     Term 117 (AT2000-0250)/Term 118 (AT2000-5250)/FB Inputs/Value Channel 29 <-> Data Pointer/RawPositionValues[28]
//     Term 117 (AT2000-0250)/Term 118 (AT2000-5250)/FB Inputs/Value Channel 30 <-> Data Pointer/RawPositionValues[29]
//     Term 117 (AT2000-0250)/Term 118 (AT2000-5250)/FB Inputs/Value Channel 31 <-> Data Pointer/RawPositionValues[30]
//     Term 117 (AT2000-0250)/Term 118 (AT2000-5250)/FB Inputs/Value Channel 32 <-> Data Pointer/RawPositionValues[31]
//   Device 24 <-> TcCOM Objects/XTS ProcessingUnit 1/Part 1/Module 60
//     Term 119 (AT2000-0250)/CC Inputs/Current actual value Ch.1 <-> Data Pointer/CurrentActualValues[0]
//     Term 119 (AT2000-0250)/CC Inputs/Current actual value Ch.10 <-> Data Pointer/CurrentActualValues[9]
//     Term 119 (AT2000-0250)/CC Inputs/Current actual value Ch.11 <-> Data Pointer/CurrentActualValues[10]
//     Term 119 (AT2000-0250)/CC Inputs/Current actual value Ch.12 <-> Data Pointer/CurrentActualValues[11]
//     Term 119 (AT2000-0250)/CC Inputs/Current actual value Ch.13 <-> Data Pointer/CurrentActualValues[12]
//     Term 119 (AT2000-0250)/CC Inputs/Current actual value Ch.14 <-> Data Pointer/CurrentActualValues[13]
//     Term 119 (AT2000-0250)/CC Inputs/Current actual value Ch.15 <-> Data Pointer/CurrentActualValues[14]
//     Term 119 (AT2000-0250)/CC Inputs/Current actual value Ch.2 <-> Data Pointer/CurrentActualValues[1]
//     Term 119 (AT2000-0250)/CC Inputs/Current actual value Ch.3 <-> Data Pointer/CurrentActualValues[2]
//     Term 119 (AT2000-0250)/CC Inputs/Current actual value Ch.4 <-> Data Pointer/CurrentActualValues[3]
//     Term 119 (AT2000-0250)/CC Inputs/Current actual value Ch.5 <-> Data Pointer/CurrentActualValues[4]
//     Term 119 (AT2000-0250)/CC Inputs/Current actual value Ch.6 <-> Data Pointer/CurrentActualValues[5]
//     Term 119 (AT2000-0250)/CC Inputs/Current actual value Ch.7 <-> Data Pointer/CurrentActualValues[6]
//     Term 119 (AT2000-0250)/CC Inputs/Current actual value Ch.8 <-> Data Pointer/CurrentActualValues[7]
//     Term 119 (AT2000-0250)/CC Inputs/Current actual value Ch.9 <-> Data Pointer/CurrentActualValues[8]
//     Term 119 (AT2000-0250)/CC Inputs/Status <-> Data Pointer/Status
//     Term 119 (AT2000-0250)/CC Outputs/Control <-> Data Pointer/Control
//     Term 119 (AT2000-0250)/CC Outputs/Current setpoint value Ch.1 <-> Data Pointer/CurrentSetpointValues[0]
//     Term 119 (AT2000-0250)/CC Outputs/Current setpoint value Ch.10 <-> Data Pointer/CurrentSetpointValues[9]
//     Term 119 (AT2000-0250)/CC Outputs/Current setpoint value Ch.11 <-> Data Pointer/CurrentSetpointValues[10]
//     Term 119 (AT2000-0250)/CC Outputs/Current setpoint value Ch.12 <-> Data Pointer/CurrentSetpointValues[11]
//     Term 119 (AT2000-0250)/CC Outputs/Current setpoint value Ch.13 <-> Data Pointer/CurrentSetpointValues[12]
//     Term 119 (AT2000-0250)/CC Outputs/Current setpoint value Ch.14 <-> Data Pointer/CurrentSetpointValues[13]
//     Term 119 (AT2000-0250)/CC Outputs/Current setpoint value Ch.15 <-> Data Pointer/CurrentSetpointValues[14]
//     Term 119 (AT2000-0250)/CC Outputs/Current setpoint value Ch.2 <-> Data Pointer/CurrentSetpointValues[1]
//     Term 119 (AT2000-0250)/CC Outputs/Current setpoint value Ch.3 <-> Data Pointer/CurrentSetpointValues[2]
//     Term 119 (AT2000-0250)/CC Outputs/Current setpoint value Ch.4 <-> Data Pointer/CurrentSetpointValues[3]
//     Term 119 (AT2000-0250)/CC Outputs/Current setpoint value Ch.5 <-> Data Pointer/CurrentSetpointValues[4]
//     Term 119 (AT2000-0250)/CC Outputs/Current setpoint value Ch.6 <-> Data Pointer/CurrentSetpointValues[5]
//     Term 119 (AT2000-0250)/CC Outputs/Current setpoint value Ch.7 <-> Data Pointer/CurrentSetpointValues[6]
//     Term 119 (AT2000-0250)/CC Outputs/Current setpoint value Ch.8 <-> Data Pointer/CurrentSetpointValues[7]
//     Term 119 (AT2000-0250)/CC Outputs/Current setpoint value Ch.9 <-> Data Pointer/CurrentSetpointValues[8]
//     Term 119 (AT2000-0250)/Term 120 (AT2000-5250)/FB Inputs/Value Channel 01 <-> Data Pointer/RawPositionValues[0]
//     Term 119 (AT2000-0250)/Term 120 (AT2000-5250)/FB Inputs/Value Channel 02 <-> Data Pointer/RawPositionValues[1]
//     Term 119 (AT2000-0250)/Term 120 (AT2000-5250)/FB Inputs/Value Channel 03 <-> Data Pointer/RawPositionValues[2]
//     Term 119 (AT2000-0250)/Term 120 (AT2000-5250)/FB Inputs/Value Channel 04 <-> Data Pointer/RawPositionValues[3]
//     Term 119 (AT2000-0250)/Term 120 (AT2000-5250)/FB Inputs/Value Channel 05 <-> Data Pointer/RawPositionValues[4]
//     Term 119 (AT2000-0250)/Term 120 (AT2000-5250)/FB Inputs/Value Channel 06 <-> Data Pointer/RawPositionValues[5]
//     Term 119 (AT2000-0250)/Term 120 (AT2000-5250)/FB Inputs/Value Channel 07 <-> Data Pointer/RawPositionValues[6]
//     Term 119 (AT2000-0250)/Term 120 (AT2000-5250)/FB Inputs/Value Channel 08 <-> Data Pointer/RawPositionValues[7]
//     Term 119 (AT2000-0250)/Term 120 (AT2000-5250)/FB Inputs/Value Channel 09 <-> Data Pointer/RawPositionValues[8]
//     Term 119 (AT2000-0250)/Term 120 (AT2000-5250)/FB Inputs/Value Channel 10 <-> Data Pointer/RawPositionValues[9]
//     Term 119 (AT2000-0250)/Term 120 (AT2000-5250)/FB Inputs/Value Channel 11 <-> Data Pointer/RawPositionValues[10]
//     Term 119 (AT2000-0250)/Term 120 (AT2000-5250)/FB Inputs/Value Channel 12 <-> Data Pointer/RawPositionValues[11]
//     Term 119 (AT2000-0250)/Term 120 (AT2000-5250)/FB Inputs/Value Channel 13 <-> Data Pointer/RawPositionValues[12]
//     Term 119 (AT2000-0250)/Term 120 (AT2000-5250)/FB Inputs/Value Channel 14 <-> Data Pointer/RawPositionValues[13]
//     Term 119 (AT2000-0250)/Term 120 (AT2000-5250)/FB Inputs/Value Channel 15 <-> Data Pointer/RawPositionValues[14]
//     Term 119 (AT2000-0250)/Term 120 (AT2000-5250)/FB Inputs/Value Channel 16 <-> Data Pointer/RawPositionValues[15]
//     Term 119 (AT2000-0250)/Term 120 (AT2000-5250)/FB Inputs/Value Channel 17 <-> Data Pointer/RawPositionValues[16]
//     Term 119 (AT2000-0250)/Term 120 (AT2000-5250)/FB Inputs/Value Channel 18 <-> Data Pointer/RawPositionValues[17]
//     Term 119 (AT2000-0250)/Term 120 (AT2000-5250)/FB Inputs/Value Channel 19 <-> Data Pointer/RawPositionValues[18]
//     Term 119 (AT2000-0250)/Term 120 (AT2000-5250)/FB Inputs/Value Channel 20 <-> Data Pointer/RawPositionValues[19]
//     Term 119 (AT2000-0250)/Term 120 (AT2000-5250)/FB Inputs/Value Channel 21 <-> Data Pointer/RawPositionValues[20]
//     Term 119 (AT2000-0250)/Term 120 (AT2000-5250)/FB Inputs/Value Channel 22 <-> Data Pointer/RawPositionValues[21]
//     Term 119 (AT2000-0250)/Term 120 (AT2000-5250)/FB Inputs/Value Channel 23 <-> Data Pointer/RawPositionValues[22]
//     Term 119 (AT2000-0250)/Term 120 (AT2000-5250)/FB Inputs/Value Channel 24 <-> Data Pointer/RawPositionValues[23]
//     Term 119 (AT2000-0250)/Term 120 (AT2000-5250)/FB Inputs/Value Channel 25 <-> Data Pointer/RawPositionValues[24]
//     Term 119 (AT2000-0250)/Term 120 (AT2000-5250)/FB Inputs/Value Channel 26 <-> Data Pointer/RawPositionValues[25]
//     Term 119 (AT2000-0250)/Term 120 (AT2000-5250)/FB Inputs/Value Channel 27 <-> Data Pointer/RawPositionValues[26]
//     Term 119 (AT2000-0250)/Term 120 (AT2000-5250)/FB Inputs/Value Channel 28 <-> Data Pointer/RawPositionValues[27]
//     Term 119 (AT2000-0250)/Term 120 (AT2000-5250)/FB Inputs/Value Channel 29 <-> Data Pointer/RawPositionValues[28]
//     Term 119 (AT2000-0250)/Term 120 (AT2000-5250)/FB Inputs/Value Channel 30 <-> Data Pointer/RawPositionValues[29]
//     Term 119 (AT2000-0250)/Term 120 (AT2000-5250)/FB Inputs/Value Channel 31 <-> Data Pointer/RawPositionValues[30]
//     Term 119 (AT2000-0250)/Term 120 (AT2000-5250)/FB Inputs/Value Channel 32 <-> Data Pointer/RawPositionValues[31]
//   Device 25 <-> TcCOM Objects/XTS ProcessingUnit 1/Part 1/Module 61
//     Term 121 (AT2002-0250)/CC Inputs/Current actual value Ch.1 <-> Data Pointer/CurrentActualValues[0]
//     Term 121 (AT2002-0250)/CC Inputs/Current actual value Ch.10 <-> Data Pointer/CurrentActualValues[9]
//     Term 121 (AT2002-0250)/CC Inputs/Current actual value Ch.11 <-> Data Pointer/CurrentActualValues[10]
//     Term 121 (AT2002-0250)/CC Inputs/Current actual value Ch.12 <-> Data Pointer/CurrentActualValues[11]
//     Term 121 (AT2002-0250)/CC Inputs/Current actual value Ch.13 <-> Data Pointer/CurrentActualValues[12]
//     Term 121 (AT2002-0250)/CC Inputs/Current actual value Ch.14 <-> Data Pointer/CurrentActualValues[13]
//     Term 121 (AT2002-0250)/CC Inputs/Current actual value Ch.15 <-> Data Pointer/CurrentActualValues[14]
//     Term 121 (AT2002-0250)/CC Inputs/Current actual value Ch.2 <-> Data Pointer/CurrentActualValues[1]
//     Term 121 (AT2002-0250)/CC Inputs/Current actual value Ch.3 <-> Data Pointer/CurrentActualValues[2]
//     Term 121 (AT2002-0250)/CC Inputs/Current actual value Ch.4 <-> Data Pointer/CurrentActualValues[3]
//     Term 121 (AT2002-0250)/CC Inputs/Current actual value Ch.5 <-> Data Pointer/CurrentActualValues[4]
//     Term 121 (AT2002-0250)/CC Inputs/Current actual value Ch.6 <-> Data Pointer/CurrentActualValues[5]
//     Term 121 (AT2002-0250)/CC Inputs/Current actual value Ch.7 <-> Data Pointer/CurrentActualValues[6]
//     Term 121 (AT2002-0250)/CC Inputs/Current actual value Ch.8 <-> Data Pointer/CurrentActualValues[7]
//     Term 121 (AT2002-0250)/CC Inputs/Current actual value Ch.9 <-> Data Pointer/CurrentActualValues[8]
//     Term 121 (AT2002-0250)/CC Inputs/Status <-> Data Pointer/Status
//     Term 121 (AT2002-0250)/CC Outputs/Control <-> Data Pointer/Control
//     Term 121 (AT2002-0250)/CC Outputs/Current setpoint value Ch.1 <-> Data Pointer/CurrentSetpointValues[0]
//     Term 121 (AT2002-0250)/CC Outputs/Current setpoint value Ch.10 <-> Data Pointer/CurrentSetpointValues[9]
//     Term 121 (AT2002-0250)/CC Outputs/Current setpoint value Ch.11 <-> Data Pointer/CurrentSetpointValues[10]
//     Term 121 (AT2002-0250)/CC Outputs/Current setpoint value Ch.12 <-> Data Pointer/CurrentSetpointValues[11]
//     Term 121 (AT2002-0250)/CC Outputs/Current setpoint value Ch.13 <-> Data Pointer/CurrentSetpointValues[12]
//     Term 121 (AT2002-0250)/CC Outputs/Current setpoint value Ch.14 <-> Data Pointer/CurrentSetpointValues[13]
//     Term 121 (AT2002-0250)/CC Outputs/Current setpoint value Ch.15 <-> Data Pointer/CurrentSetpointValues[14]
//     Term 121 (AT2002-0250)/CC Outputs/Current setpoint value Ch.2 <-> Data Pointer/CurrentSetpointValues[1]
//     Term 121 (AT2002-0250)/CC Outputs/Current setpoint value Ch.3 <-> Data Pointer/CurrentSetpointValues[2]
//     Term 121 (AT2002-0250)/CC Outputs/Current setpoint value Ch.4 <-> Data Pointer/CurrentSetpointValues[3]
//     Term 121 (AT2002-0250)/CC Outputs/Current setpoint value Ch.5 <-> Data Pointer/CurrentSetpointValues[4]
//     Term 121 (AT2002-0250)/CC Outputs/Current setpoint value Ch.6 <-> Data Pointer/CurrentSetpointValues[5]
//     Term 121 (AT2002-0250)/CC Outputs/Current setpoint value Ch.7 <-> Data Pointer/CurrentSetpointValues[6]
//     Term 121 (AT2002-0250)/CC Outputs/Current setpoint value Ch.8 <-> Data Pointer/CurrentSetpointValues[7]
//     Term 121 (AT2002-0250)/CC Outputs/Current setpoint value Ch.9 <-> Data Pointer/CurrentSetpointValues[8]
//     Term 121 (AT2002-0250)/Term 122 (AT2002-5250)/FB Inputs/Value Channel 01 <-> Data Pointer/RawPositionValues[0]
//     Term 121 (AT2002-0250)/Term 122 (AT2002-5250)/FB Inputs/Value Channel 02 <-> Data Pointer/RawPositionValues[1]
//     Term 121 (AT2002-0250)/Term 122 (AT2002-5250)/FB Inputs/Value Channel 03 <-> Data Pointer/RawPositionValues[2]
//     Term 121 (AT2002-0250)/Term 122 (AT2002-5250)/FB Inputs/Value Channel 04 <-> Data Pointer/RawPositionValues[3]
//     Term 121 (AT2002-0250)/Term 122 (AT2002-5250)/FB Inputs/Value Channel 05 <-> Data Pointer/RawPositionValues[4]
//     Term 121 (AT2002-0250)/Term 122 (AT2002-5250)/FB Inputs/Value Channel 06 <-> Data Pointer/RawPositionValues[5]
//     Term 121 (AT2002-0250)/Term 122 (AT2002-5250)/FB Inputs/Value Channel 07 <-> Data Pointer/RawPositionValues[6]
//     Term 121 (AT2002-0250)/Term 122 (AT2002-5250)/FB Inputs/Value Channel 08 <-> Data Pointer/RawPositionValues[7]
//     Term 121 (AT2002-0250)/Term 122 (AT2002-5250)/FB Inputs/Value Channel 09 <-> Data Pointer/RawPositionValues[8]
//     Term 121 (AT2002-0250)/Term 122 (AT2002-5250)/FB Inputs/Value Channel 10 <-> Data Pointer/RawPositionValues[9]
//     Term 121 (AT2002-0250)/Term 122 (AT2002-5250)/FB Inputs/Value Channel 11 <-> Data Pointer/RawPositionValues[10]
//     Term 121 (AT2002-0250)/Term 122 (AT2002-5250)/FB Inputs/Value Channel 12 <-> Data Pointer/RawPositionValues[11]
//     Term 121 (AT2002-0250)/Term 122 (AT2002-5250)/FB Inputs/Value Channel 13 <-> Data Pointer/RawPositionValues[12]
//     Term 121 (AT2002-0250)/Term 122 (AT2002-5250)/FB Inputs/Value Channel 14 <-> Data Pointer/RawPositionValues[13]
//     Term 121 (AT2002-0250)/Term 122 (AT2002-5250)/FB Inputs/Value Channel 15 <-> Data Pointer/RawPositionValues[14]
//     Term 121 (AT2002-0250)/Term 122 (AT2002-5250)/FB Inputs/Value Channel 16 <-> Data Pointer/RawPositionValues[15]
//     Term 121 (AT2002-0250)/Term 122 (AT2002-5250)/FB Inputs/Value Channel 17 <-> Data Pointer/RawPositionValues[16]
//     Term 121 (AT2002-0250)/Term 122 (AT2002-5250)/FB Inputs/Value Channel 18 <-> Data Pointer/RawPositionValues[17]
//     Term 121 (AT2002-0250)/Term 122 (AT2002-5250)/FB Inputs/Value Channel 19 <-> Data Pointer/RawPositionValues[18]
//     Term 121 (AT2002-0250)/Term 122 (AT2002-5250)/FB Inputs/Value Channel 20 <-> Data Pointer/RawPositionValues[19]
//     Term 121 (AT2002-0250)/Term 122 (AT2002-5250)/FB Inputs/Value Channel 21 <-> Data Pointer/RawPositionValues[20]
//     Term 121 (AT2002-0250)/Term 122 (AT2002-5250)/FB Inputs/Value Channel 22 <-> Data Pointer/RawPositionValues[21]
//     Term 121 (AT2002-0250)/Term 122 (AT2002-5250)/FB Inputs/Value Channel 23 <-> Data Pointer/RawPositionValues[22]
//     Term 121 (AT2002-0250)/Term 122 (AT2002-5250)/FB Inputs/Value Channel 24 <-> Data Pointer/RawPositionValues[23]
//     Term 121 (AT2002-0250)/Term 122 (AT2002-5250)/FB Inputs/Value Channel 25 <-> Data Pointer/RawPositionValues[24]
//     Term 121 (AT2002-0250)/Term 122 (AT2002-5250)/FB Inputs/Value Channel 26 <-> Data Pointer/RawPositionValues[25]
//     Term 121 (AT2002-0250)/Term 122 (AT2002-5250)/FB Inputs/Value Channel 27 <-> Data Pointer/RawPositionValues[26]
//     Term 121 (AT2002-0250)/Term 122 (AT2002-5250)/FB Inputs/Value Channel 28 <-> Data Pointer/RawPositionValues[27]
//     Term 121 (AT2002-0250)/Term 122 (AT2002-5250)/FB Inputs/Value Channel 29 <-> Data Pointer/RawPositionValues[28]
//     Term 121 (AT2002-0250)/Term 122 (AT2002-5250)/FB Inputs/Value Channel 30 <-> Data Pointer/RawPositionValues[29]
//     Term 121 (AT2002-0250)/Term 122 (AT2002-5250)/FB Inputs/Value Channel 31 <-> Data Pointer/RawPositionValues[30]
//     Term 121 (AT2002-0250)/Term 122 (AT2002-5250)/FB Inputs/Value Channel 32 <-> Data Pointer/RawPositionValues[31]
//   Device 25 <-> TcCOM Objects/XTS ProcessingUnit 1/Part 1/Module 62
//     Term 123 (AT2000-0250)/CC Inputs/Current actual value Ch.1 <-> Data Pointer/CurrentActualValues[0]
//     Term 123 (AT2000-0250)/CC Inputs/Current actual value Ch.10 <-> Data Pointer/CurrentActualValues[9]
//     Term 123 (AT2000-0250)/CC Inputs/Current actual value Ch.11 <-> Data Pointer/CurrentActualValues[10]
//     Term 123 (AT2000-0250)/CC Inputs/Current actual value Ch.12 <-> Data Pointer/CurrentActualValues[11]
//     Term 123 (AT2000-0250)/CC Inputs/Current actual value Ch.13 <-> Data Pointer/CurrentActualValues[12]
//     Term 123 (AT2000-0250)/CC Inputs/Current actual value Ch.14 <-> Data Pointer/CurrentActualValues[13]
//     Term 123 (AT2000-0250)/CC Inputs/Current actual value Ch.15 <-> Data Pointer/CurrentActualValues[14]
//     Term 123 (AT2000-0250)/CC Inputs/Current actual value Ch.2 <-> Data Pointer/CurrentActualValues[1]
//     Term 123 (AT2000-0250)/CC Inputs/Current actual value Ch.3 <-> Data Pointer/CurrentActualValues[2]
//     Term 123 (AT2000-0250)/CC Inputs/Current actual value Ch.4 <-> Data Pointer/CurrentActualValues[3]
//     Term 123 (AT2000-0250)/CC Inputs/Current actual value Ch.5 <-> Data Pointer/CurrentActualValues[4]
//     Term 123 (AT2000-0250)/CC Inputs/Current actual value Ch.6 <-> Data Pointer/CurrentActualValues[5]
//     Term 123 (AT2000-0250)/CC Inputs/Current actual value Ch.7 <-> Data Pointer/CurrentActualValues[6]
//     Term 123 (AT2000-0250)/CC Inputs/Current actual value Ch.8 <-> Data Pointer/CurrentActualValues[7]
//     Term 123 (AT2000-0250)/CC Inputs/Current actual value Ch.9 <-> Data Pointer/CurrentActualValues[8]
//     Term 123 (AT2000-0250)/CC Inputs/Status <-> Data Pointer/Status
//     Term 123 (AT2000-0250)/CC Outputs/Control <-> Data Pointer/Control
//     Term 123 (AT2000-0250)/CC Outputs/Current setpoint value Ch.1 <-> Data Pointer/CurrentSetpointValues[0]
//     Term 123 (AT2000-0250)/CC Outputs/Current setpoint value Ch.10 <-> Data Pointer/CurrentSetpointValues[9]
//     Term 123 (AT2000-0250)/CC Outputs/Current setpoint value Ch.11 <-> Data Pointer/CurrentSetpointValues[10]
//     Term 123 (AT2000-0250)/CC Outputs/Current setpoint value Ch.12 <-> Data Pointer/CurrentSetpointValues[11]
//     Term 123 (AT2000-0250)/CC Outputs/Current setpoint value Ch.13 <-> Data Pointer/CurrentSetpointValues[12]
//     Term 123 (AT2000-0250)/CC Outputs/Current setpoint value Ch.14 <-> Data Pointer/CurrentSetpointValues[13]
//     Term 123 (AT2000-0250)/CC Outputs/Current setpoint value Ch.15 <-> Data Pointer/CurrentSetpointValues[14]
//     Term 123 (AT2000-0250)/CC Outputs/Current setpoint value Ch.2 <-> Data Pointer/CurrentSetpointValues[1]
//     Term 123 (AT2000-0250)/CC Outputs/Current setpoint value Ch.3 <-> Data Pointer/CurrentSetpointValues[2]
//     Term 123 (AT2000-0250)/CC Outputs/Current setpoint value Ch.4 <-> Data Pointer/CurrentSetpointValues[3]
//     Term 123 (AT2000-0250)/CC Outputs/Current setpoint value Ch.5 <-> Data Pointer/CurrentSetpointValues[4]
//     Term 123 (AT2000-0250)/CC Outputs/Current setpoint value Ch.6 <-> Data Pointer/CurrentSetpointValues[5]
//     Term 123 (AT2000-0250)/CC Outputs/Current setpoint value Ch.7 <-> Data Pointer/CurrentSetpointValues[6]
//     Term 123 (AT2000-0250)/CC Outputs/Current setpoint value Ch.8 <-> Data Pointer/CurrentSetpointValues[7]
//     Term 123 (AT2000-0250)/CC Outputs/Current setpoint value Ch.9 <-> Data Pointer/CurrentSetpointValues[8]
//     Term 123 (AT2000-0250)/Term 124 (AT2000-5250)/FB Inputs/Value Channel 01 <-> Data Pointer/RawPositionValues[0]
//     Term 123 (AT2000-0250)/Term 124 (AT2000-5250)/FB Inputs/Value Channel 02 <-> Data Pointer/RawPositionValues[1]
//     Term 123 (AT2000-0250)/Term 124 (AT2000-5250)/FB Inputs/Value Channel 03 <-> Data Pointer/RawPositionValues[2]
//     Term 123 (AT2000-0250)/Term 124 (AT2000-5250)/FB Inputs/Value Channel 04 <-> Data Pointer/RawPositionValues[3]
//     Term 123 (AT2000-0250)/Term 124 (AT2000-5250)/FB Inputs/Value Channel 05 <-> Data Pointer/RawPositionValues[4]
//     Term 123 (AT2000-0250)/Term 124 (AT2000-5250)/FB Inputs/Value Channel 06 <-> Data Pointer/RawPositionValues[5]
//     Term 123 (AT2000-0250)/Term 124 (AT2000-5250)/FB Inputs/Value Channel 07 <-> Data Pointer/RawPositionValues[6]
//     Term 123 (AT2000-0250)/Term 124 (AT2000-5250)/FB Inputs/Value Channel 08 <-> Data Pointer/RawPositionValues[7]
//     Term 123 (AT2000-0250)/Term 124 (AT2000-5250)/FB Inputs/Value Channel 09 <-> Data Pointer/RawPositionValues[8]
//     Term 123 (AT2000-0250)/Term 124 (AT2000-5250)/FB Inputs/Value Channel 10 <-> Data Pointer/RawPositionValues[9]
//     Term 123 (AT2000-0250)/Term 124 (AT2000-5250)/FB Inputs/Value Channel 11 <-> Data Pointer/RawPositionValues[10]
//     Term 123 (AT2000-0250)/Term 124 (AT2000-5250)/FB Inputs/Value Channel 12 <-> Data Pointer/RawPositionValues[11]
//     Term 123 (AT2000-0250)/Term 124 (AT2000-5250)/FB Inputs/Value Channel 13 <-> Data Pointer/RawPositionValues[12]
//     Term 123 (AT2000-0250)/Term 124 (AT2000-5250)/FB Inputs/Value Channel 14 <-> Data Pointer/RawPositionValues[13]
//     Term 123 (AT2000-0250)/Term 124 (AT2000-5250)/FB Inputs/Value Channel 15 <-> Data Pointer/RawPositionValues[14]
//     Term 123 (AT2000-0250)/Term 124 (AT2000-5250)/FB Inputs/Value Channel 16 <-> Data Pointer/RawPositionValues[15]
//     Term 123 (AT2000-0250)/Term 124 (AT2000-5250)/FB Inputs/Value Channel 17 <-> Data Pointer/RawPositionValues[16]
//     Term 123 (AT2000-0250)/Term 124 (AT2000-5250)/FB Inputs/Value Channel 18 <-> Data Pointer/RawPositionValues[17]
//     Term 123 (AT2000-0250)/Term 124 (AT2000-5250)/FB Inputs/Value Channel 19 <-> Data Pointer/RawPositionValues[18]
//     Term 123 (AT2000-0250)/Term 124 (AT2000-5250)/FB Inputs/Value Channel 20 <-> Data Pointer/RawPositionValues[19]
//     Term 123 (AT2000-0250)/Term 124 (AT2000-5250)/FB Inputs/Value Channel 21 <-> Data Pointer/RawPositionValues[20]
//     Term 123 (AT2000-0250)/Term 124 (AT2000-5250)/FB Inputs/Value Channel 22 <-> Data Pointer/RawPositionValues[21]
//     Term 123 (AT2000-0250)/Term 124 (AT2000-5250)/FB Inputs/Value Channel 23 <-> Data Pointer/RawPositionValues[22]
//     Term 123 (AT2000-0250)/Term 124 (AT2000-5250)/FB Inputs/Value Channel 24 <-> Data Pointer/RawPositionValues[23]
//     Term 123 (AT2000-0250)/Term 124 (AT2000-5250)/FB Inputs/Value Channel 25 <-> Data Pointer/RawPositionValues[24]
//     Term 123 (AT2000-0250)/Term 124 (AT2000-5250)/FB Inputs/Value Channel 26 <-> Data Pointer/RawPositionValues[25]
//     Term 123 (AT2000-0250)/Term 124 (AT2000-5250)/FB Inputs/Value Channel 27 <-> Data Pointer/RawPositionValues[26]
//     Term 123 (AT2000-0250)/Term 124 (AT2000-5250)/FB Inputs/Value Channel 28 <-> Data Pointer/RawPositionValues[27]
//     Term 123 (AT2000-0250)/Term 124 (AT2000-5250)/FB Inputs/Value Channel 29 <-> Data Pointer/RawPositionValues[28]
//     Term 123 (AT2000-0250)/Term 124 (AT2000-5250)/FB Inputs/Value Channel 30 <-> Data Pointer/RawPositionValues[29]
//     Term 123 (AT2000-0250)/Term 124 (AT2000-5250)/FB Inputs/Value Channel 31 <-> Data Pointer/RawPositionValues[30]
//     Term 123 (AT2000-0250)/Term 124 (AT2000-5250)/FB Inputs/Value Channel 32 <-> Data Pointer/RawPositionValues[31]
//   Device 25 <-> TcCOM Objects/XTS ProcessingUnit 1/Part 1/Module 63
//     Term 125 (AT2000-0250)/CC Inputs/Current actual value Ch.1 <-> Data Pointer/CurrentActualValues[0]
//     Term 125 (AT2000-0250)/CC Inputs/Current actual value Ch.10 <-> Data Pointer/CurrentActualValues[9]
//     Term 125 (AT2000-0250)/CC Inputs/Current actual value Ch.11 <-> Data Pointer/CurrentActualValues[10]
//     Term 125 (AT2000-0250)/CC Inputs/Current actual value Ch.12 <-> Data Pointer/CurrentActualValues[11]
//     Term 125 (AT2000-0250)/CC Inputs/Current actual value Ch.13 <-> Data Pointer/CurrentActualValues[12]
//     Term 125 (AT2000-0250)/CC Inputs/Current actual value Ch.14 <-> Data Pointer/CurrentActualValues[13]
//     Term 125 (AT2000-0250)/CC Inputs/Current actual value Ch.15 <-> Data Pointer/CurrentActualValues[14]
//     Term 125 (AT2000-0250)/CC Inputs/Current actual value Ch.2 <-> Data Pointer/CurrentActualValues[1]
//     Term 125 (AT2000-0250)/CC Inputs/Current actual value Ch.3 <-> Data Pointer/CurrentActualValues[2]
//     Term 125 (AT2000-0250)/CC Inputs/Current actual value Ch.4 <-> Data Pointer/CurrentActualValues[3]
//     Term 125 (AT2000-0250)/CC Inputs/Current actual value Ch.5 <-> Data Pointer/CurrentActualValues[4]
//     Term 125 (AT2000-0250)/CC Inputs/Current actual value Ch.6 <-> Data Pointer/CurrentActualValues[5]
//     Term 125 (AT2000-0250)/CC Inputs/Current actual value Ch.7 <-> Data Pointer/CurrentActualValues[6]
//     Term 125 (AT2000-0250)/CC Inputs/Current actual value Ch.8 <-> Data Pointer/CurrentActualValues[7]
//     Term 125 (AT2000-0250)/CC Inputs/Current actual value Ch.9 <-> Data Pointer/CurrentActualValues[8]
//     Term 125 (AT2000-0250)/CC Inputs/Status <-> Data Pointer/Status
//     Term 125 (AT2000-0250)/CC Outputs/Control <-> Data Pointer/Control
//     Term 125 (AT2000-0250)/CC Outputs/Current setpoint value Ch.1 <-> Data Pointer/CurrentSetpointValues[0]
//     Term 125 (AT2000-0250)/CC Outputs/Current setpoint value Ch.10 <-> Data Pointer/CurrentSetpointValues[9]
//     Term 125 (AT2000-0250)/CC Outputs/Current setpoint value Ch.11 <-> Data Pointer/CurrentSetpointValues[10]
//     Term 125 (AT2000-0250)/CC Outputs/Current setpoint value Ch.12 <-> Data Pointer/CurrentSetpointValues[11]
//     Term 125 (AT2000-0250)/CC Outputs/Current setpoint value Ch.13 <-> Data Pointer/CurrentSetpointValues[12]
//     Term 125 (AT2000-0250)/CC Outputs/Current setpoint value Ch.14 <-> Data Pointer/CurrentSetpointValues[13]
//     Term 125 (AT2000-0250)/CC Outputs/Current setpoint value Ch.15 <-> Data Pointer/CurrentSetpointValues[14]
//     Term 125 (AT2000-0250)/CC Outputs/Current setpoint value Ch.2 <-> Data Pointer/CurrentSetpointValues[1]
//     Term 125 (AT2000-0250)/CC Outputs/Current setpoint value Ch.3 <-> Data Pointer/CurrentSetpointValues[2]
//     Term 125 (AT2000-0250)/CC Outputs/Current setpoint value Ch.4 <-> Data Pointer/CurrentSetpointValues[3]
//     Term 125 (AT2000-0250)/CC Outputs/Current setpoint value Ch.5 <-> Data Pointer/CurrentSetpointValues[4]
//     Term 125 (AT2000-0250)/CC Outputs/Current setpoint value Ch.6 <-> Data Pointer/CurrentSetpointValues[5]
//     Term 125 (AT2000-0250)/CC Outputs/Current setpoint value Ch.7 <-> Data Pointer/CurrentSetpointValues[6]
//     Term 125 (AT2000-0250)/CC Outputs/Current setpoint value Ch.8 <-> Data Pointer/CurrentSetpointValues[7]
//     Term 125 (AT2000-0250)/CC Outputs/Current setpoint value Ch.9 <-> Data Pointer/CurrentSetpointValues[8]
//     Term 125 (AT2000-0250)/Term 126 (AT2000-5250)/FB Inputs/Value Channel 01 <-> Data Pointer/RawPositionValues[0]
//     Term 125 (AT2000-0250)/Term 126 (AT2000-5250)/FB Inputs/Value Channel 02 <-> Data Pointer/RawPositionValues[1]
//     Term 125 (AT2000-0250)/Term 126 (AT2000-5250)/FB Inputs/Value Channel 03 <-> Data Pointer/RawPositionValues[2]
//     Term 125 (AT2000-0250)/Term 126 (AT2000-5250)/FB Inputs/Value Channel 04 <-> Data Pointer/RawPositionValues[3]
//     Term 125 (AT2000-0250)/Term 126 (AT2000-5250)/FB Inputs/Value Channel 05 <-> Data Pointer/RawPositionValues[4]
//     Term 125 (AT2000-0250)/Term 126 (AT2000-5250)/FB Inputs/Value Channel 06 <-> Data Pointer/RawPositionValues[5]
//     Term 125 (AT2000-0250)/Term 126 (AT2000-5250)/FB Inputs/Value Channel 07 <-> Data Pointer/RawPositionValues[6]
//     Term 125 (AT2000-0250)/Term 126 (AT2000-5250)/FB Inputs/Value Channel 08 <-> Data Pointer/RawPositionValues[7]
//     Term 125 (AT2000-0250)/Term 126 (AT2000-5250)/FB Inputs/Value Channel 09 <-> Data Pointer/RawPositionValues[8]
//     Term 125 (AT2000-0250)/Term 126 (AT2000-5250)/FB Inputs/Value Channel 10 <-> Data Pointer/RawPositionValues[9]
//     Term 125 (AT2000-0250)/Term 126 (AT2000-5250)/FB Inputs/Value Channel 11 <-> Data Pointer/RawPositionValues[10]
//     Term 125 (AT2000-0250)/Term 126 (AT2000-5250)/FB Inputs/Value Channel 12 <-> Data Pointer/RawPositionValues[11]
//     Term 125 (AT2000-0250)/Term 126 (AT2000-5250)/FB Inputs/Value Channel 13 <-> Data Pointer/RawPositionValues[12]
//     Term 125 (AT2000-0250)/Term 126 (AT2000-5250)/FB Inputs/Value Channel 14 <-> Data Pointer/RawPositionValues[13]
//     Term 125 (AT2000-0250)/Term 126 (AT2000-5250)/FB Inputs/Value Channel 15 <-> Data Pointer/RawPositionValues[14]
//     Term 125 (AT2000-0250)/Term 126 (AT2000-5250)/FB Inputs/Value Channel 16 <-> Data Pointer/RawPositionValues[15]
//     Term 125 (AT2000-0250)/Term 126 (AT2000-5250)/FB Inputs/Value Channel 17 <-> Data Pointer/RawPositionValues[16]
//     Term 125 (AT2000-0250)/Term 126 (AT2000-5250)/FB Inputs/Value Channel 18 <-> Data Pointer/RawPositionValues[17]
//     Term 125 (AT2000-0250)/Term 126 (AT2000-5250)/FB Inputs/Value Channel 19 <-> Data Pointer/RawPositionValues[18]
//     Term 125 (AT2000-0250)/Term 126 (AT2000-5250)/FB Inputs/Value Channel 20 <-> Data Pointer/RawPositionValues[19]
//     Term 125 (AT2000-0250)/Term 126 (AT2000-5250)/FB Inputs/Value Channel 21 <-> Data Pointer/RawPositionValues[20]
//     Term 125 (AT2000-0250)/Term 126 (AT2000-5250)/FB Inputs/Value Channel 22 <-> Data Pointer/RawPositionValues[21]
